LIN {X 0,Y 368.88,Z 241.032,A -85,B 0,C 180,E1 -12741.361,E2 -12741.361} C_VEL
LIN {X 0,Y 368.933,Z 241.028,A -85,B 0,C 180,E1 -12745.14,E2 -12745.14} C_VEL
LIN {X 0,Y 368.915,Z 241.029,A -85,B 0,C 180,E1 -12749.039,E2 -12749.039} C_VEL
LIN {X 0,Y 368.907,Z 241.03,A -85,B 0,C 180,E1 -12751.552,E2 -12751.552} C_VEL
LIN {X 0,Y 368.92,Z 241.03,A -85,B 0,C 180,E1 -12755.216,E2 -12755.216} C_VEL
LIN {X 0,Y 368.917,Z 241.033,A -85,B 0,C 180,E1 -12758.975,E2 -12758.975} C_VEL
LIN {X 0,Y 368.933,Z 241.027,A -85,B 0,C 180,E1 -12762.256,E2 -12762.256} C_VEL
LIN {X 0,Y 369.039,Z 241.014,A -85,B 0,C 180,E1 -12766.216,E2 -12766.216} C_VEL
LIN {X 0,Y 369.049,Z 241.013,A -85,B 0,C 180,E1 -12770.125,E2 -12770.125} C_VEL
LIN {X 0,Y 369.165,Z 240.997,A -85,B 0,C 180,E1 -12773.434,E2 -12773.434} C_VEL
LIN {X 0,Y 369.287,Z 240.984,A -85,B 0,C 180,E1 -12777.812,E2 -12777.812} C_VEL
LIN {X 0,Y 369.437,Z 240.962,A -85,B 0,C 180,E1 -12779.993,E2 -12779.993} C_VEL
LIN {X 0,Y 369.298,Z 240.98,A -85,B 0,C 180,E1 -12782.174,E2 -12782.174} C_VEL
LIN {X 0,Y 369.16,Z 241,A -85,B 0,C 180,E1 -12786.551,E2 -12786.551} C_VEL
LIN {X 0,Y 369.099,Z 241.008,A -85,B 0,C 180,E1 -12788.754,E2 -12788.754} C_VEL
LIN {X 0,Y 368.987,Z 241.022,A -85,B 0,C 180,E1 -12792.086,E2 -12792.086} C_VEL
LIN {X 0,Y 368.969,Z 241.027,A -85,B 0,C 180,E1 -12795.457,E2 -12795.457} C_VEL
LIN {X 0,Y 368.973,Z 241.053,A -85,B 0,C 180,E1 -12799.137,E2 -12799.137} C_VEL
LIN {X 0,Y 369.122,Z 241.853,A -85,B 0,C 180,E1 -12799.454,E2 -12799.454} C_VEL
LIN {X 0,Y 371.497,Z 252.434,A -85,B 0,C 180,E1 -12802.223,E2 -12802.223} C_VEL
LIN {X 0,Y 372.489,Z 258.071,A -85,B 0,C 180,E1 -12803.627,E2 -12803.627} C_VEL
LIN {X 0,Y 372.536,Z 259.043,A -85,B 0,C 180,E1 -12803.809,E2 -12803.809} C_VEL
LIN {X 0,Y 376.937,Z 279.442,A -85,B 0,C 180,E1 -12804.621,E2 -12804.621} C_VEL
LIN {X 0,Y 378.226,Z 287.075,A -85,B 0,C 180,E1 -12804.882,E2 -12804.882} C_VEL
LIN {X 0,Y 376.362,Z 367.62,A -85,B 0,C 180,E1 -12806.593,E2 -12806.593} C_VEL
LIN {X 0,Y 375.694,Z 381.568,A -85,B 0,C 180,E1 -12807.118,E2 -12807.118} C_VEL
LIN {X 0,Y 374.985,Z 393.464,A -85,B 0,C 180,E1 -12807.778,E2 -12807.778} C_VEL
LIN {X 0,Y 374.005,Z 405.344,A -85,B 0,C 180,E1 -12808.66,E2 -12808.66} C_VEL
LIN {X 0,Y 372.898,Z 416.825,A -85,B 0,C 180,E1 -12809.756,E2 -12809.756} C_VEL
LIN {X 0,Y 371.777,Z 427.103,A -85,B 0,C 180,E1 -12810.983,E2 -12810.983} C_VEL
LIN {X 0,Y 370.754,Z 436.401,A -85,B 0,C 180,E1 -12812.367,E2 -12812.367} C_VEL
LIN {X 0,Y 369.821,Z 444.095,A -85,B 0,C 180,E1 -12813.759,E2 -12813.759} C_VEL
LIN {X 0,Y 369.08,Z 450.98,A -85,B 0,C 180,E1 -12815.281,E2 -12815.281} C_VEL
LIN {X 0,Y 368.38,Z 457.744,A -85,B 0,C 180,E1 -12817.156,E2 -12817.156} C_VEL
LIN {X 0,Y 367.823,Z 462.959,A -85,B 0,C 180,E1 -12819.077,E2 -12819.077} C_VEL
LIN {X 0,Y 367.554,Z 465.968,A -85,B 0,C 180,E1 -12820.537,E2 -12820.537} C_VEL
LIN {X 0,Y 367.345,Z 468.186,A -85,B 0,C 180,E1 -12822.024,E2 -12822.024} C_VEL
LIN {X 0,Y 367.242,Z 469.646,A -85,B 0,C 180,E1 -12823.532,E2 -12823.532} C_VEL
LIN {X 0,Y 367.153,Z 470.359,A -85,B 0,C 180,E1 -12825.079,E2 -12825.079} C_VEL
LIN {X 0,Y 367.105,Z 470.265,A -85,B 0,C 180,E1 -12826.661,E2 -12826.661} C_VEL
LIN {X 0,Y 367.181,Z 469.289,A -85,B 0,C 180,E1 -12828.271,E2 -12828.271} C_VEL
LIN {X 0,Y 367.289,Z 467.345,A -85,B 0,C 180,E1 -12829.926,E2 -12829.926} C_VEL
LIN {X 0,Y 367.518,Z 464.352,A -85,B 0,C 180,E1 -12831.615,E2 -12831.615} C_VEL
LIN {X 0,Y 367.894,Z 459.129,A -85,B 0,C 180,E1 -12833.689,E2 -12833.689} C_VEL
LIN {X 0,Y 368.411,Z 453.179,A -85,B 0,C 180,E1 -12835.46,E2 -12835.46} C_VEL
LIN {X 0,Y 368.975,Z 446.012,A -85,B 0,C 180,E1 -12837.149,E2 -12837.149} C_VEL
LIN {X 0,Y 369.786,Z 437.345,A -85,B 0,C 180,E1 -12838.767,E2 -12838.767} C_VEL
LIN {X 0,Y 370.61,Z 428.223,A -85,B 0,C 180,E1 -12840.149,E2 -12840.149} C_VEL
LIN {X 0,Y 371.441,Z 418.859,A -85,B 0,C 180,E1 -12841.309,E2 -12841.309} C_VEL
LIN {X 0,Y 372.382,Z 407.076,A -85,B 0,C 180,E1 -12842.48,E2 -12842.48} C_VEL
LIN {X 0,Y 373.302,Z 394.459,A -85,B 0,C 180,E1 -12843.443,E2 -12843.443} C_VEL
LIN {X 0,Y 373.975,Z 382.071,A -85,B 0,C 180,E1 -12844.149,E2 -12844.149} C_VEL
LIN {X 0,Y 374.556,Z 368.268,A -85,B 0,C 180,E1 -12844.678,E2 -12844.678} C_VEL
LIN {X 0,Y 375.164,Z 336.229,A -85,B 0,C 180,E1 -12845.369,E2 -12845.369} C_VEL
LIN {X 0,Y 376.006,Z 284.873,A -85,B 0,C 180,E1 -12846.423,E2 -12846.423} C_VEL
LIN {X 0,Y 371.483,Z 259.793,A -85,B 0,C 180,E1 -12847.219,E2 -12847.219} C_VEL
LIN {X 0,Y 371.535,Z 258.335,A -85,B 0,C 180,E1 -12847.48,E2 -12847.48} C_VEL
LIN {X 0,Y 371.55,Z 254.8,A -85,B 0,C 180,E1 -12848.409,E2 -12848.409} C_VEL
LIN {X 0,Y 369.334,Z 242.98,A -85,B 0,C 180,E1 -12851.704,E2 -12851.704} C_VEL
LIN {X 0,Y 368.973,Z 241.05,A -85,B 0,C 180,E1 -12852.346,E2 -12852.346} C_VEL
LIN {X 0,Y 368.965,Z 241.024,A -85,B 0,C 180,E1 -12856.227,E2 -12856.227} C_VEL
LIN {X 0,Y 369,Z 241.018,A -85,B 0,C 180,E1 -12860.132,E2 -12860.132} C_VEL
LIN {X 0,Y 369.091,Z 241.008,A -85,B 0,C 180,E1 -12862.342,E2 -12862.342} C_VEL
LIN {X 0,Y 369.078,Z 241.01,A -85,B 0,C 180,E1 -12864.539,E2 -12864.539} C_VEL
LIN {X 0,Y 369.252,Z 240.985,A -85,B 0,C 180,E1 -12867.82,E2 -12867.82} C_VEL
LIN {X 0,Y 369.388,Z 240.968,A -85,B 0,C 180,E1 -12870.002,E2 -12870.002} C_VEL
LIN {X 0,Y 369.088,Z 241.011,A -85,B 0,C 180,E1 -12873.277,E2 -12873.277} C_VEL
LIN {X 0,Y 369.061,Z 241.013,A -85,B 0,C 180,E1 -12873.418,E2 -12873.418} C_VEL
LIN {X 0,Y 368.32,Z 241.102,A -85,B 0,C 180,E1 -12874.329,E2 -12874.329} C_VEL
LIN {X 0,Y 365.557,Z 241.446,A -85,B 0,C 180,E1 -12875.813,E2 -12875.813} C_VEL
LIN {X 0,Y 363.239,Z 241.738,A -85,B 0,C 180,E1 -12877.013,E2 -12877.013} C_VEL
LIN {X 0,Y 362.191,Z 241.866,A -85,B 0,C 180,E1 -12877.939,E2 -12877.939} C_VEL
LIN {X 0,Y 362.073,Z 241.879,A -85,B 0,C 180,E1 -12878.252,E2 -12878.252} C_VEL
LIN {X 0,Y 361.9,Z 241.901,A -85,B 0,C 180,E1 -12882.336,E2 -12882.336} C_VEL
LIN {X 0,Y 361.896,Z 241.901,A -85,B 0,C 180,E1 -12884.625,E2 -12884.625} C_VEL
LIN {X 0,Y 361.892,Z 241.904,A -85,B 0,C 180,E1 -12888.104,E2 -12888.104} C_VEL
LIN {X 0,Y 361.822,Z 241.917,A -85,B 0,C 180,E1 -12891.659,E2 -12891.659} C_VEL
LIN {X 0,Y 361.869,Z 241.906,A -85,B 0,C 180,E1 -12895.296,E2 -12895.296} C_VEL
LIN {X 0,Y 361.866,Z 241.91,A -85,B 0,C 180,E1 -12897.784,E2 -12897.784} C_VEL
LIN {X 0,Y 361.806,Z 241.915,A -85,B 0,C 180,E1 -12901.634,E2 -12901.634} C_VEL
LIN {X 0,Y 361.824,Z 241.91,A -85,B 0,C 180,E1 -12905.352,E2 -12905.352} C_VEL
LIN {X 0,Y 361.827,Z 241.911,A -85,B 0,C 180,E1 -12909.035,E2 -12909.035} C_VEL
LIN {X 0,Y 361.843,Z 241.915,A -85,B 0,C 180,E1 -12912.448,E2 -12912.448} C_VEL
LIN {X 0,Y 361.891,Z 241.903,A -85,B 0,C 180,E1 -12915.937,E2 -12915.937} C_VEL
LIN {X 0,Y 361.87,Z 241.906,A -85,B 0,C 180,E1 -12919.24,E2 -12919.24} C_VEL
LIN {X 0,Y 361.845,Z 241.913,A -85,B 0,C 180,E1 -12922.992,E2 -12922.992} C_VEL
LIN {X 0,Y 361.831,Z 241.913,A -85,B 0,C 180,E1 -12926.64,E2 -12926.64} C_VEL
LIN {X 0,Y 361.849,Z 241.908,A -85,B 0,C 180,E1 -12929.681,E2 -12929.681} C_VEL
LIN {X 0,Y 361.934,Z 241.9,A -85,B 0,C 180,E1 -12933.484,E2 -12933.484} C_VEL
LIN {X 0,Y 361.864,Z 241.911,A -85,B 0,C 180,E1 -12937.153,E2 -12937.153} C_VEL
LIN {X 0,Y 361.872,Z 241.905,A -85,B 0,C 180,E1 -12940.731,E2 -12940.731} C_VEL
LIN {X 0,Y 361.935,Z 241.897,A -85,B 0,C 180,E1 -12944.234,E2 -12944.234} C_VEL
LIN {X 0,Y 361.994,Z 241.889,A -85,B 0,C 180,E1 -12946.536,E2 -12946.536} C_VEL
LIN {X 0,Y 362.026,Z 241.89,A -85,B 0,C 180,E1 -12949.946,E2 -12949.946} C_VEL
LIN {X 0,Y 362.124,Z 241.875,A -85,B 0,C 180,E1 -12953.321,E2 -12953.321} C_VEL
LIN {X 0,Y 362.275,Z 241.859,A -85,B 0,C 180,E1 -12957.784,E2 -12957.784} C_VEL
LIN {X 0,Y 362.271,Z 241.861,A -85,B 0,C 180,E1 -12962.231,E2 -12962.231} C_VEL
LIN {X 0,Y 362.133,Z 241.874,A -85,B 0,C 180,E1 -12966.694,E2 -12966.694} C_VEL
LIN {X 0,Y 362.01,Z 241.89,A -85,B 0,C 180,E1 -12970.069,E2 -12970.069} C_VEL
LIN {X 0,Y 362.015,Z 241.888,A -85,B 0,C 180,E1 -12973.904,E2 -12973.904} C_VEL
LIN {X 0,Y 361.946,Z 241.899,A -85,B 0,C 180,E1 -12976.94,E2 -12976.94} C_VEL
LIN {X 0,Y 361.902,Z 241.904,A -85,B 0,C 180,E1 -12980.466,E2 -12980.466} C_VEL
LIN {X 0,Y 361.915,Z 241.899,A -85,B 0,C 180,E1 -12984.117,E2 -12984.117} C_VEL
LIN {X 0,Y 361.856,Z 241.907,A -85,B 0,C 180,E1 -12987.79,E2 -12987.79} C_VEL
LIN {X 0,Y 361.87,Z 241.91,A -85,B 0,C 180,E1 -12991.289,E2 -12991.289} C_VEL
LIN {X 0,Y 361.876,Z 241.904,A -85,B 0,C 180,E1 -12994.284,E2 -12994.284} C_VEL
LIN {X 0,Y 361.883,Z 241.909,A -85,B 0,C 180,E1 -12997.225,E2 -12997.225} C_VEL
LIN {X 0,Y 361.833,Z 241.91,A -85,B 0,C 180,E1 -13000.753,E2 -13000.753} C_VEL
LIN {X 0,Y 361.81,Z 241.912,A -85,B 0,C 180,E1 -13004.376,E2 -13004.376} C_VEL
LIN {X 0,Y 361.837,Z 241.915,A -85,B 0,C 180,E1 -13007.574,E2 -13007.574} C_VEL
LIN {X 0,Y 361.866,Z 241.909,A -85,B 0,C 180,E1 -13011.573,E2 -13011.573} C_VEL
LIN {X 0,Y 361.894,Z 241.902,A -85,B 0,C 180,E1 -13014.658,E2 -13014.658} C_VEL
LIN {X 0,Y 361.862,Z 241.912,A -85,B 0,C 180,E1 -13018.371,E2 -13018.371} C_VEL
LIN {X 0,Y 361.923,Z 241.987,A -85,B 0,C 180,E1 -13021.432,E2 -13021.432} C_VEL
LIN {X 0,Y 364.248,Z 253.417,A -85,B 0,C 180,E1 -13024.575,E2 -13024.575} C_VEL
LIN {X 0,Y 365.247,Z 259.524,A -85,B 0,C 180,E1 -13026.165,E2 -13026.165} C_VEL
LIN {X 0,Y 364.377,Z 268.912,A -85,B 0,C 180,E1 -13028.396,E2 -13028.396} C_VEL
LIN {X 0,Y 365.363,Z 275.194,A -85,B 0,C 180,E1 -13028.638,E2 -13028.638} C_VEL
LIN {X 0,Y 369.292,Z 299.895,A -85,B 0,C 180,E1 -13029.389,E2 -13029.389} C_VEL
LIN {X 0,Y 367.75,Z 377.611,A -85,B 0,C 180,E1 -13031.04,E2 -13031.04} C_VEL
LIN {X 0,Y 367.12,Z 391.044,A -85,B 0,C 180,E1 -13031.549,E2 -13031.549} C_VEL
LIN {X 0,Y 366.383,Z 403.845,A -85,B 0,C 180,E1 -13032.269,E2 -13032.269} C_VEL
LIN {X 0,Y 365.338,Z 416.379,A -85,B 0,C 180,E1 -13033.227,E2 -13033.227} C_VEL
LIN {X 0,Y 364.389,Z 427.609,A -85,B 0,C 180,E1 -13034.333,E2 -13034.333} C_VEL
LIN {X 0,Y 363.664,Z 436.712,A -85,B 0,C 180,E1 -13035.448,E2 -13035.448} C_VEL
LIN {X 0,Y 362.744,Z 446.03,A -85,B 0,C 180,E1 -13036.839,E2 -13036.839} C_VEL
LIN {X 0,Y 361.838,Z 455.084,A -85,B 0,C 180,E1 -13038.515,E2 -13038.515} C_VEL
LIN {X 0,Y 361.216,Z 462.362,A -85,B 0,C 180,E1 -13040.196,E2 -13040.196} C_VEL
LIN {X 0,Y 360.843,Z 467.262,A -85,B 0,C 180,E1 -13041.599,E2 -13041.599} C_VEL
LIN {X 0,Y 360.529,Z 472.006,A -85,B 0,C 180,E1 -13043.281,E2 -13043.281} C_VEL
LIN {X 0,Y 360.361,Z 475.609,A -85,B 0,C 180,E1 -13044.963,E2 -13044.963} C_VEL
LIN {X 0,Y 360.284,Z 478.174,A -85,B 0,C 180,E1 -13046.643,E2 -13046.643} C_VEL
LIN {X 0,Y 360.234,Z 479.363,A -85,B 0,C 180,E1 -13047.762,E2 -13047.762} C_VEL
LIN {X 0,Y 360.259,Z 480.099,A -85,B 0,C 180,E1 -13048.88,E2 -13048.88} C_VEL
LIN {X 0,Y 360.285,Z 480.438,A -85,B 0,C 180,E1 -13049.998,E2 -13049.998} C_VEL
LIN {X 0,Y 360.257,Z 480.382,A -85,B 0,C 180,E1 -13051.116,E2 -13051.116} C_VEL
LIN {X 0,Y 360.232,Z 479.92,A -85,B 0,C 180,E1 -13052.234,E2 -13052.234} C_VEL
LIN {X 0,Y 360.284,Z 479.017,A -85,B 0,C 180,E1 -13053.353,E2 -13053.353} C_VEL
LIN {X 0,Y 360.37,Z 477.711,A -85,B 0,C 180,E1 -13054.472,E2 -13054.472} C_VEL
LIN {X 0,Y 360.474,Z 475.098,A -85,B 0,C 180,E1 -13056.076,E2 -13056.076} C_VEL
LIN {X 0,Y 360.771,Z 471.152,A -85,B 0,C 180,E1 -13057.835,E2 -13057.835} C_VEL
LIN {X 0,Y 361.265,Z 466.224,A -85,B 0,C 180,E1 -13059.516,E2 -13059.516} C_VEL
LIN {X 0,Y 361.94,Z 460.024,A -85,B 0,C 180,E1 -13061.194,E2 -13061.194} C_VEL
LIN {X 0,Y 362.832,Z 452.335,A -85,B 0,C 180,E1 -13062.869,E2 -13062.869} C_VEL
LIN {X 0,Y 364.083,Z 442.682,A -85,B 0,C 180,E1 -13064.531,E2 -13064.531} C_VEL
LIN {X 0,Y 365.093,Z 432.754,A -85,B 0,C 180,E1 -13065.919,E2 -13065.919} C_VEL
LIN {X 0,Y 366.141,Z 423.009,A -85,B 0,C 180,E1 -13067.019,E2 -13067.019} C_VEL
LIN {X 0,Y 367.4,Z 410.731,A -85,B 0,C 180,E1 -13068.108,E2 -13068.108} C_VEL
LIN {X 0,Y 368.393,Z 399.904,A -85,B 0,C 180,E1 -13068.85,E2 -13068.85} C_VEL
LIN {X 0,Y 369.213,Z 386.728,A -85,B 0,C 180,E1 -13069.528,E2 -13069.528} C_VEL
LIN {X 0,Y 369.858,Z 373.38,A -85,B 0,C 180,E1 -13069.962,E2 -13069.962} C_VEL
LIN {X 0,Y 371.447,Z 299.693,A -85,B 0,C 180,E1 -13071.55,E2 -13071.55} C_VEL
LIN {X 0,Y 367.766,Z 278.61,A -85,B 0,C 180,E1 -13072.318,E2 -13072.318} C_VEL
LIN {X 0,Y 365.474,Z 268.168,A -85,B 0,C 180,E1 -13072.764,E2 -13072.764} C_VEL
LIN {X 0,Y 365.983,Z 262.373,A -85,B 0,C 180,E1 -13074.081,E2 -13074.081} C_VEL
LIN {X 0,Y 364.601,Z 253.875,A -85,B 0,C 180,E1 -13076.315,E2 -13076.315} C_VEL
LIN {X 0,Y 362.372,Z 244.187,A -85,B 0,C 180,E1 -13079.001,E2 -13079.001} C_VEL
LIN {X 0,Y 361.899,Z 241.952,A -85,B 0,C 180,E1 -13079.72,E2 -13079.72} C_VEL
LIN {X 0,Y 361.87,Z 241.91,A -85,B 0,C 180,E1 -13083.365,E2 -13083.365} C_VEL
LIN {X 0,Y 361.873,Z 241.909,A -85,B 0,C 180,E1 -13087.014,E2 -13087.014} C_VEL
LIN {X 0,Y 361.819,Z 241.913,A -85,B 0,C 180,E1 -13090.746,E2 -13090.746} C_VEL
LIN {X 0,Y 361.818,Z 241.917,A -85,B 0,C 180,E1 -13094.365,E2 -13094.365} C_VEL
LIN {X 0,Y 361.828,Z 241.913,A -85,B 0,C 180,E1 -13097.566,E2 -13097.566} C_VEL
LIN {X 0,Y 361.846,Z 241.909,A -85,B 0,C 180,E1 -13101.566,E2 -13101.566} C_VEL
LIN {X 0,Y 361.873,Z 241.909,A -85,B 0,C 180,E1 -13104.651,E2 -13104.651} C_VEL
LIN {X 0,Y 361.84,Z 241.914,A -85,B 0,C 180,E1 -13108.365,E2 -13108.365} C_VEL
LIN {X 0,Y 361.85,Z 241.91,A -85,B 0,C 180,E1 -13110.945,E2 -13110.945} C_VEL
LIN {X 0,Y 361.878,Z 241.906,A -85,B 0,C 180,E1 -13114.7,E2 -13114.7} C_VEL
LIN {X 0,Y 361.85,Z 241.908,A -85,B 0,C 180,E1 -13118.338,E2 -13118.338} C_VEL
LIN {X 0,Y 361.89,Z 241.903,A -85,B 0,C 180,E1 -13122.091,E2 -13122.091} C_VEL
LIN {X 0,Y 361.98,Z 241.894,A -85,B 0,C 180,E1 -13126.102,E2 -13126.102} C_VEL
LIN {X 0,Y 361.986,Z 241.893,A -85,B 0,C 180,E1 -13129.93,E2 -13129.93} C_VEL
LIN {X 0,Y 362.127,Z 241.875,A -85,B 0,C 180,E1 -13133.306,E2 -13133.306} C_VEL
LIN {X 0,Y 362.25,Z 241.86,A -85,B 0,C 180,E1 -13137.769,E2 -13137.769} C_VEL
LIN {X 0,Y 362.386,Z 241.84,A -85,B 0,C 180,E1 -13139.993,E2 -13139.993} C_VEL
LIN {X 0,Y 362.261,Z 241.856,A -85,B 0,C 180,E1 -13142.216,E2 -13142.216} C_VEL
LIN {X 0,Y 362.124,Z 241.877,A -85,B 0,C 180,E1 -13146.679,E2 -13146.679} C_VEL
LIN {X 0,Y 362.011,Z 241.891,A -85,B 0,C 180,E1 -13150.054,E2 -13150.054} C_VEL
LIN {X 0,Y 361.97,Z 241.898,A -85,B 0,C 180,E1 -13153.892,E2 -13153.892} C_VEL
LIN {X 0,Y 361.938,Z 241.899,A -85,B 0,C 180,E1 -13157.933,E2 -13157.933} C_VEL
LIN {X 0,Y 361.962,Z 242.037,A -85,B 0,C 180,E1 -13158.75,E2 -13158.75} C_VEL
LIN {X 0,Y 364.246,Z 252.021,A -85,B 0,C 180,E1 -13161.497,E2 -13161.497} C_VEL
LIN {X 0,Y 365.659,Z 258.999,A -85,B 0,C 180,E1 -13163.27,E2 -13163.27} C_VEL
LIN {X 0,Y 367.677,Z 267.137,A -85,B 0,C 180,E1 -13163.657,E2 -13163.657} C_VEL
LIN {X 0,Y 371.681,Z 286.962,A -85,B 0,C 180,E1 -13164.423,E2 -13164.423} C_VEL
LIN {X 0,Y 369.795,Z 367.824,A -85,B 0,C 180,E1 -13166.183,E2 -13166.183} C_VEL
LIN {X 0,Y 369.116,Z 381.433,A -85,B 0,C 180,E1 -13166.703,E2 -13166.703} C_VEL
LIN {X 0,Y 368.336,Z 393.75,A -85,B 0,C 180,E1 -13167.397,E2 -13167.397} C_VEL
LIN {X 0,Y 367.268,Z 406.035,A -85,B 0,C 180,E1 -13168.333,E2 -13168.333} C_VEL
LIN {X 0,Y 366.128,Z 417.468,A -85,B 0,C 180,E1 -13169.454,E2 -13169.454} C_VEL
LIN {X 0,Y 364.962,Z 427.464,A -85,B 0,C 180,E1 -13170.68,E2 -13170.68} C_VEL
LIN {X 0,Y 363.751,Z 437.747,A -85,B 0,C 180,E1 -13172.265,E2 -13172.265} C_VEL
LIN {X 0,Y 362.704,Z 446.064,A -85,B 0,C 180,E1 -13173.857,E2 -13173.857} C_VEL
LIN {X 0,Y 361.852,Z 453.395,A -85,B 0,C 180,E1 -13175.627,E2 -13175.627} C_VEL
LIN {X 0,Y 361.303,Z 458.357,A -85,B 0,C 180,E1 -13177.11,E2 -13177.11} C_VEL
LIN {X 0,Y 360.789,Z 462.891,A -85,B 0,C 180,E1 -13178.818,E2 -13178.818} C_VEL
LIN {X 0,Y 360.463,Z 466.266,A -85,B 0,C 180,E1 -13180.505,E2 -13180.505} C_VEL
LIN {X 0,Y 360.25,Z 468.601,A -85,B 0,C 180,E1 -13182.159,E2 -13182.159} C_VEL
LIN {X 0,Y 360.121,Z 469.991,A -85,B 0,C 180,E1 -13183.777,E2 -13183.777} C_VEL
LIN {X 0,Y 360.043,Z 470.506,A -85,B 0,C 180,E1 -13185.358,E2 -13185.358} C_VEL
LIN {X 0,Y 360.018,Z 470.24,A -85,B 0,C 180,E1 -13186.906,E2 -13186.906} C_VEL
LIN {X 0,Y 360.083,Z 469.235,A -85,B 0,C 180,E1 -13188.428,E2 -13188.428} C_VEL
LIN {X 0,Y 360.295,Z 466.376,A -85,B 0,C 180,E1 -13190.629,E2 -13190.629} C_VEL
LIN {X 0,Y 360.625,Z 461.794,A -85,B 0,C 180,E1 -13192.836,E2 -13192.836} C_VEL
LIN {X 0,Y 361.112,Z 456.042,A -85,B 0,C 180,E1 -13194.808,E2 -13194.808} C_VEL
LIN {X 0,Y 361.719,Z 449.081,A -85,B 0,C 180,E1 -13196.645,E2 -13196.645} C_VEL
LIN {X 0,Y 362.308,Z 442.248,A -85,B 0,C 180,E1 -13198.092,E2 -13198.092} C_VEL
LIN {X 0,Y 363.179,Z 433.295,A -85,B 0,C 180,E1 -13199.635,E2 -13199.635} C_VEL
LIN {X 0,Y 364.096,Z 423.384,A -85,B 0,C 180,E1 -13201.02,E2 -13201.02} C_VEL
LIN {X 0,Y 365.122,Z 412.051,A -85,B 0,C 180,E1 -13202.28,E2 -13202.28} C_VEL
LIN {X 0,Y 366.059,Z 399.91,A -85,B 0,C 180,E1 -13203.337,E2 -13203.337} C_VEL
LIN {X 0,Y 366.872,Z 387.097,A -85,B 0,C 180,E1 -13204.18,E2 -13204.18} C_VEL
LIN {X 0,Y 367.518,Z 373.473,A -85,B 0,C 180,E1 -13204.808,E2 -13204.808} C_VEL
LIN {X 0,Y 367.969,Z 359.673,A -85,B 0,C 180,E1 -13205.197,E2 -13205.197} C_VEL
LIN {X 0,Y 369.272,Z 285.9,A -85,B 0,C 180,E1 -13206.742,E2 -13206.742} C_VEL
LIN {X 0,Y 364.621,Z 260.016,A -85,B 0,C 180,E1 -13207.573,E2 -13207.573} C_VEL
LIN {X 0,Y 364.641,Z 258.567,A -85,B 0,C 180,E1 -13207.82,E2 -13207.82} C_VEL
LIN {X 0,Y 364.184,Z 253.951,A -85,B 0,C 180,E1 -13209.086,E2 -13209.086} C_VEL
LIN {X 0,Y 361.936,Z 242.118,A -85,B 0,C 180,E1 -13212.486,E2 -13212.486} C_VEL
LIN {X 0,Y 361.926,Z 241.9,A -85,B 0,C 180,E1 -13216.101,E2 -13216.101} C_VEL
LIN {X 0,Y 361.964,Z 241.893,A -85,B 0,C 180,E1 -13219.938,E2 -13219.938} C_VEL
LIN {X 0,Y 362.095,Z 241.878,A -85,B 0,C 180,E1 -13223.314,E2 -13223.314} C_VEL
LIN {X 0,Y 362.218,Z 241.861,A -85,B 0,C 180,E1 -13227.778,E2 -13227.778} C_VEL
LIN {X 0,Y 362.358,Z 241.844,A -85,B 0,C 180,E1 -13230.002,E2 -13230.002} C_VEL
LIN {X 0,Y 362.218,Z 241.861,A -85,B 0,C 180,E1 -13232.226,E2 -13232.226} C_VEL
LIN {X 0,Y 362.098,Z 241.878,A -85,B 0,C 180,E1 -13236.689,E2 -13236.689} C_VEL
LIN {X 0,Y 362.073,Z 241.879,A -85,B 0,C 180,E1 -13238.252,E2 -13238.252} C_VEL
LIN {X 0,Y 361.302,Z 241.981,A -85,B 0,C 180,E1 -13239.18,E2 -13239.18} C_VEL
LIN {X 0,Y 358.365,Z 242.342,A -85,B 0,C 180,E1 -13240.688,E2 -13240.688} C_VEL
LIN {X 0,Y 355.945,Z 242.645,A -85,B 0,C 180,E1 -13241.908,E2 -13241.908} C_VEL
LIN {X 0,Y 354.928,Z 242.771,A -85,B 0,C 180,E1 -13242.853,E2 -13242.853} C_VEL
LIN {X 0,Y 354.854,Z 242.778,A -85,B 0,C 180,E1 -13243.173,E2 -13243.173} C_VEL
LIN {X 0,Y 354.824,Z 242.784,A -85,B 0,C 180,E1 -13246.101,E2 -13246.101} C_VEL
LIN {X 0,Y 354.837,Z 242.781,A -85,B 0,C 180,E1 -13248.477,E2 -13248.477} C_VEL
LIN {X 0,Y 354.769,Z 242.792,A -85,B 0,C 180,E1 -13252.112,E2 -13252.112} C_VEL
LIN {X 0,Y 354.841,Z 242.787,A -85,B 0,C 180,E1 -13255.834,E2 -13255.834} C_VEL
LIN {X 0,Y 354.8,Z 242.789,A -85,B 0,C 180,E1 -13259.685,E2 -13259.685} C_VEL
LIN {X 0,Y 354.78,Z 242.79,A -85,B 0,C 180,E1 -13263.689,E2 -13263.689} C_VEL
LIN {X 0,Y 354.75,Z 242.796,A -85,B 0,C 180,E1 -13266.467,E2 -13266.467} C_VEL
LIN {X 0,Y 354.779,Z 242.788,A -85,B 0,C 180,E1 -13269.431,E2 -13269.431} C_VEL
LIN {X 0,Y 354.799,Z 242.788,A -85,B 0,C 180,E1 -13272.884,E2 -13272.884} C_VEL
LIN {X 0,Y 354.829,Z 242.784,A -85,B 0,C 180,E1 -13276.127,E2 -13276.127} C_VEL
LIN {X 0,Y 354.821,Z 242.784,A -85,B 0,C 180,E1 -13279.197,E2 -13279.197} C_VEL
LIN {X 0,Y 354.784,Z 242.79,A -85,B 0,C 180,E1 -13282.41,E2 -13282.41} C_VEL
LIN {X 0,Y 354.784,Z 242.794,A -85,B 0,C 180,E1 -13284.95,E2 -13284.95} C_VEL
LIN {X 0,Y 354.768,Z 242.791,A -85,B 0,C 180,E1 -13288.414,E2 -13288.414} C_VEL
LIN {X 0,Y 354.825,Z 242.784,A -85,B 0,C 180,E1 -13291.627,E2 -13291.627} C_VEL
LIN {X 0,Y 354.88,Z 242.775,A -85,B 0,C 180,E1 -13294.181,E2 -13294.181} C_VEL
LIN {X 0,Y 354.801,Z 242.786,A -85,B 0,C 180,E1 -13297.901,E2 -13297.901} C_VEL
LIN {X 0,Y 354.88,Z 242.777,A -85,B 0,C 180,E1 -13301.917,E2 -13301.917} C_VEL
LIN {X 0,Y 354.937,Z 242.771,A -85,B 0,C 180,E1 -13305.99,E2 -13305.99} C_VEL
LIN {X 0,Y 354.973,Z 242.771,A -85,B 0,C 180,E1 -13309.744,E2 -13309.744} C_VEL
LIN {X 0,Y 355.09,Z 242.75,A -85,B 0,C 180,E1 -13313.188,E2 -13313.188} C_VEL
LIN {X 0,Y 355.238,Z 242.735,A -85,B 0,C 180,E1 -13317.74,E2 -13317.74} C_VEL
LIN {X 0,Y 355.176,Z 242.739,A -85,B 0,C 180,E1 -13321.141,E2 -13321.141} C_VEL
LIN {X 0,Y 355.234,Z 242.737,A -85,B 0,C 180,E1 -13322.275,E2 -13322.275} C_VEL
LIN {X 0,Y 355.099,Z 242.75,A -85,B 0,C 180,E1 -13326.827,E2 -13326.827} C_VEL
LIN {X 0,Y 354.967,Z 242.77,A -85,B 0,C 180,E1 -13330.271,E2 -13330.271} C_VEL
LIN {X 0,Y 354.959,Z 242.767,A -85,B 0,C 180,E1 -13334.024,E2 -13334.024} C_VEL
LIN {X 0,Y 354.909,Z 242.773,A -85,B 0,C 180,E1 -13338.098,E2 -13338.098} C_VEL
LIN {X 0,Y 354.833,Z 242.782,A -85,B 0,C 180,E1 -13342.113,E2 -13342.113} C_VEL
LIN {X 0,Y 354.869,Z 242.78,A -85,B 0,C 180,E1 -13344.582,E2 -13344.582} C_VEL
LIN {X 0,Y 354.819,Z 242.784,A -85,B 0,C 180,E1 -13348.39,E2 -13348.39} C_VEL
LIN {X 0,Y 354.809,Z 242.784,A -85,B 0,C 180,E1 -13352.337,E2 -13352.337} C_VEL
LIN {X 0,Y 354.844,Z 242.782,A -85,B 0,C 180,E1 -13355.702,E2 -13355.702} C_VEL
LIN {X 0,Y 354.793,Z 242.793,A -85,B 0,C 180,E1 -13359.415,E2 -13359.415} C_VEL
LIN {X 0,Y 354.785,Z 242.788,A -85,B 0,C 180,E1 -13362.865,E2 -13362.865} C_VEL
LIN {X 0,Y 354.768,Z 242.791,A -85,B 0,C 180,E1 -13366.102,E2 -13366.102} C_VEL
LIN {X 0,Y 354.785,Z 242.789,A -85,B 0,C 180,E1 -13369.177,E2 -13369.177} C_VEL
LIN {X 0,Y 354.823,Z 242.784,A -85,B 0,C 180,E1 -13372.406,E2 -13372.406} C_VEL
LIN {X 0,Y 354.832,Z 242.781,A -85,B 0,C 180,E1 -13374.941,E2 -13374.941} C_VEL
LIN {X 0,Y 354.818,Z 242.79,A -85,B 0,C 180,E1 -13378.406,E2 -13378.406} C_VEL
LIN {X 0,Y 354.884,Z 242.917,A -85,B 0,C 180,E1 -13381.167,E2 -13381.167} C_VEL
LIN {X 0,Y 357.197,Z 254.28,A -85,B 0,C 180,E1 -13384.349,E2 -13384.349} C_VEL
LIN {X 0,Y 358.252,Z 260.391,A -85,B 0,C 180,E1 -13385.978,E2 -13385.978} C_VEL
LIN {X 0,Y 357.499,Z 268.825,A -85,B 0,C 180,E1 -13388.023,E2 -13388.023} C_VEL
LIN {X 0,Y 359.02,Z 278.379,A -85,B 0,C 180,E1 -13388.369,E2 -13388.369} C_VEL
LIN {X 0,Y 362.548,Z 300.61,A -85,B 0,C 180,E1 -13389.062,E2 -13389.062} C_VEL
LIN {X 0,Y 360.955,Z 376.817,A -85,B 0,C 180,E1 -13390.706,E2 -13390.706} C_VEL
LIN {X 0,Y 360.321,Z 390.465,A -85,B 0,C 180,E1 -13391.225,E2 -13391.225} C_VEL
LIN {X 0,Y 359.564,Z 402.895,A -85,B 0,C 180,E1 -13391.922,E2 -13391.922} C_VEL
LIN {X 0,Y 358.665,Z 414.041,A -85,B 0,C 180,E1 -13392.758,E2 -13392.758} C_VEL
LIN {X 0,Y 357.651,Z 425.676,A -85,B 0,C 180,E1 -13393.883,E2 -13393.883} C_VEL
LIN {X 0,Y 356.761,Z 436.177,A -85,B 0,C 180,E1 -13395.16,E2 -13395.16} C_VEL
LIN {X 0,Y 355.787,Z 445.597,A -85,B 0,C 180,E1 -13396.577,E2 -13396.577} C_VEL
LIN {X 0,Y 354.846,Z 454.711,A -85,B 0,C 180,E1 -13398.285,E2 -13398.285} C_VEL
LIN {X 0,Y 354.193,Z 462.046,A -85,B 0,C 180,E1 -13400,E2 -13400} C_VEL
LIN {X 0,Y 353.802,Z 466.985,A -85,B 0,C 180,E1 -13401.43,E2 -13401.43} C_VEL
LIN {X 0,Y 353.446,Z 471.769,A -85,B 0,C 180,E1 -13403.146,E2 -13403.146} C_VEL
LIN {X 0,Y 353.268,Z 475.408,A -85,B 0,C 180,E1 -13404.862,E2 -13404.862} C_VEL
LIN {X 0,Y 353.208,Z 478.007,A -85,B 0,C 180,E1 -13406.576,E2 -13406.576} C_VEL
LIN {X 0,Y 353.145,Z 479.22,A -85,B 0,C 180,E1 -13407.717,E2 -13407.717} C_VEL
LIN {X 0,Y 353.158,Z 479.978,A -85,B 0,C 180,E1 -13408.858,E2 -13408.858} C_VEL
LIN {X 0,Y 353.186,Z 480.331,A -85,B 0,C 180,E1 -13409.998,E2 -13409.998} C_VEL
LIN {X 0,Y 353.157,Z 480.289,A -85,B 0,C 180,E1 -13411.138,E2 -13411.138} C_VEL
LIN {X 0,Y 353.143,Z 479.849,A -85,B 0,C 180,E1 -13412.279,E2 -13412.279} C_VEL
LIN {X 0,Y 353.209,Z 478.964,A -85,B 0,C 180,E1 -13413.42,E2 -13413.42} C_VEL
LIN {X 0,Y 353.287,Z 477.671,A -85,B 0,C 180,E1 -13414.562,E2 -13414.562} C_VEL
LIN {X 0,Y 353.389,Z 475.372,A -85,B 0,C 180,E1 -13416.048,E2 -13416.048} C_VEL
LIN {X 0,Y 353.726,Z 471.178,A -85,B 0,C 180,E1 -13417.992,E2 -13417.992} C_VEL
LIN {X 0,Y 354.231,Z 466.293,A -85,B 0,C 180,E1 -13419.707,E2 -13419.707} C_VEL
LIN {X 0,Y 354.938,Z 460.14,A -85,B 0,C 180,E1 -13421.418,E2 -13421.418} C_VEL
LIN {X 0,Y 355.919,Z 452.498,A -85,B 0,C 180,E1 -13423.123,E2 -13423.123} C_VEL
LIN {X 0,Y 357.004,Z 444.693,A -85,B 0,C 180,E1 -13424.534,E2 -13424.534} C_VEL
LIN {X 0,Y 358.035,Z 435.188,A -85,B 0,C 180,E1 -13425.949,E2 -13425.949} C_VEL
LIN {X 0,Y 359.253,Z 424.67,A -85,B 0,C 180,E1 -13427.209,E2 -13427.209} C_VEL
LIN {X 0,Y 360.569,Z 412.998,A -85,B 0,C 180,E1 -13428.316,E2 -13428.316} C_VEL
LIN {X 0,Y 361.574,Z 401.726,A -85,B 0,C 180,E1 -13429.145,E2 -13429.145} C_VEL
LIN {X 0,Y 362.572,Z 387.774,A -85,B 0,C 180,E1 -13429.901,E2 -13429.901} C_VEL
LIN {X 0,Y 363.237,Z 375.474,A -85,B 0,C 180,E1 -13430.342,E2 -13430.342} C_VEL
LIN {X 0,Y 365.02,Z 300.893,A -85,B 0,C 180,E1 -13431.992,E2 -13431.992} C_VEL
LIN {X 0,Y 361.842,Z 282.186,A -85,B 0,C 180,E1 -13432.685,E2 -13432.685} C_VEL
LIN {X 0,Y 358.768,Z 267.831,A -85,B 0,C 180,E1 -13433.327,E2 -13433.327} C_VEL
LIN {X 0,Y 359.017,Z 262.654,A -85,B 0,C 180,E1 -13434.579,E2 -13434.579} C_VEL
LIN {X 0,Y 357.117,Z 252.395,A -85,B 0,C 180,E1 -13437.371,E2 -13437.371} C_VEL
LIN {X 0,Y 354.842,Z 242.847,A -85,B 0,C 180,E1 -13440.209,E2 -13440.209} C_VEL
LIN {X 0,Y 354.819,Z 242.789,A -85,B 0,C 180,E1 -13443.698,E2 -13443.698} C_VEL
LIN {X 0,Y 354.806,Z 242.791,A -85,B 0,C 180,E1 -13446.456,E2 -13446.456} C_VEL
LIN {X 0,Y 354.779,Z 242.791,A -85,B 0,C 180,E1 -13449.408,E2 -13449.408} C_VEL
LIN {X 0,Y 354.789,Z 242.788,A -85,B 0,C 180,E1 -13452.861,E2 -13452.861} C_VEL
LIN {X 0,Y 354.768,Z 242.792,A -85,B 0,C 180,E1 -13456.097,E2 -13456.097} C_VEL
LIN {X 0,Y 354.768,Z 242.793,A -85,B 0,C 180,E1 -13459.17,E2 -13459.17} C_VEL
LIN {X 0,Y 354.803,Z 242.791,A -85,B 0,C 180,E1 -13462.399,E2 -13462.399} C_VEL
LIN {X 0,Y 354.811,Z 242.789,A -85,B 0,C 180,E1 -13464.934,E2 -13464.934} C_VEL
LIN {X 0,Y 354.796,Z 242.792,A -85,B 0,C 180,E1 -13468.399,E2 -13468.399} C_VEL
LIN {X 0,Y 354.789,Z 242.789,A -85,B 0,C 180,E1 -13471.607,E2 -13471.607} C_VEL
LIN {X 0,Y 354.841,Z 242.783,A -85,B 0,C 180,E1 -13475.416,E2 -13475.416} C_VEL
LIN {X 0,Y 354.815,Z 242.788,A -85,B 0,C 180,E1 -13479.106,E2 -13479.106} C_VEL
LIN {X 0,Y 354.833,Z 242.787,A -85,B 0,C 180,E1 -13482.71,E2 -13482.71} C_VEL
LIN {X 0,Y 354.939,Z 242.771,A -85,B 0,C 180,E1 -13486.248,E2 -13486.248} C_VEL
LIN {X 0,Y 354.943,Z 242.771,A -85,B 0,C 180,E1 -13489.728,E2 -13489.728} C_VEL
LIN {X 0,Y 355.091,Z 242.753,A -85,B 0,C 180,E1 -13493.173,E2 -13493.173} C_VEL
LIN {X 0,Y 355.213,Z 242.736,A -85,B 0,C 180,E1 -13497.725,E2 -13497.725} C_VEL
LIN {X 0,Y 355.336,Z 242.718,A -85,B 0,C 180,E1 -13499.993,E2 -13499.993} C_VEL
LIN {X 0,Y 355.224,Z 242.733,A -85,B 0,C 180,E1 -13502.26,E2 -13502.26} C_VEL
LIN {X 0,Y 355.09,Z 242.753,A -85,B 0,C 180,E1 -13506.812,E2 -13506.812} C_VEL
LIN {X 0,Y 354.958,Z 242.769,A -85,B 0,C 180,E1 -13510.256,E2 -13510.256} C_VEL
LIN {X 0,Y 354.915,Z 242.777,A -85,B 0,C 180,E1 -13514.012,E2 -13514.012} C_VEL
LIN {X 0,Y 354.914,Z 242.876,A -85,B 0,C 180,E1 -13518.214,E2 -13518.214} C_VEL
LIN {X 0,Y 357.207,Z 252.764,A -85,B 0,C 180,E1 -13521.033,E2 -13521.033} C_VEL
LIN {X 0,Y 358.569,Z 259.336,A -85,B 0,C 180,E1 -13522.723,E2 -13522.723} C_VEL
LIN {X 0,Y 360.426,Z 264.571,A -85,B 0,C 180,E1 -13523.02,E2 -13523.02} C_VEL
LIN {X 0,Y 364.798,Z 285.505,A -85,B 0,C 180,E1 -13523.876,E2 -13523.876} C_VEL
LIN {X 0,Y 365.282,Z 289.608,A -85,B 0,C 180,E1 -13524.011,E2 -13524.011} C_VEL
LIN {X 0,Y 363.266,Z 368.071,A -85,B 0,C 180,E1 -13525.756,E2 -13525.756} C_VEL
LIN {X 0,Y 362.524,Z 381.844,A -85,B 0,C 180,E1 -13526.295,E2 -13526.295} C_VEL
LIN {X 0,Y 361.695,Z 394.113,A -85,B 0,C 180,E1 -13527.007,E2 -13527.007} C_VEL
LIN {X 0,Y 360.715,Z 405.301,A -85,B 0,C 180,E1 -13527.868,E2 -13527.868} C_VEL
LIN {X 0,Y 359.629,Z 415.405,A -85,B 0,C 180,E1 -13528.844,E2 -13528.844} C_VEL
LIN {X 0,Y 358.275,Z 426.752,A -85,B 0,C 180,E1 -13530.215,E2 -13530.215} C_VEL
LIN {X 0,Y 357.2,Z 435.764,A -85,B 0,C 180,E1 -13531.58,E2 -13531.58} C_VEL
LIN {X 0,Y 356.011,Z 444.468,A -85,B 0,C 180,E1 -13533.205,E2 -13533.205} C_VEL
LIN {X 0,Y 355.044,Z 452.243,A -85,B 0,C 180,E1 -13535.021,E2 -13535.021} C_VEL
LIN {X 0,Y 354.278,Z 458.724,A -85,B 0,C 180,E1 -13536.97,E2 -13536.97} C_VEL
LIN {X 0,Y 353.781,Z 462.91,A -85,B 0,C 180,E1 -13538.584,E2 -13538.584} C_VEL
LIN {X 0,Y 353.439,Z 466.117,A -85,B 0,C 180,E1 -13540.187,E2 -13540.187} C_VEL
LIN {X 0,Y 353.27,Z 467.427,A -85,B 0,C 180,E1 -13541.02,E2 -13541.02} C_VEL
LIN {X 0,Y 353.125,Z 469.241,A -85,B 0,C 180,E1 -13542.579,E2 -13542.579} C_VEL
LIN {X 0,Y 352.996,Z 470.336,A -85,B 0,C 180,E1 -13544.217,E2 -13544.217} C_VEL
LIN {X 0,Y 352.943,Z 470.608,A -85,B 0,C 180,E1 -13545.822,E2 -13545.822} C_VEL
LIN {X 0,Y 352.945,Z 470.077,A -85,B 0,C 180,E1 -13547.441,E2 -13547.441} C_VEL
LIN {X 0,Y 353.027,Z 468.61,A -85,B 0,C 180,E1 -13549.14,E2 -13549.14} C_VEL
LIN {X 0,Y 353.244,Z 466.147,A -85,B 0,C 180,E1 -13550.872,E2 -13550.872} C_VEL
LIN {X 0,Y 353.496,Z 462.524,A -85,B 0,C 180,E1 -13552.662,E2 -13552.662} C_VEL
LIN {X 0,Y 353.915,Z 457.559,A -85,B 0,C 180,E1 -13554.487,E2 -13554.487} C_VEL
LIN {X 0,Y 354.513,Z 450.992,A -85,B 0,C 180,E1 -13556.35,E2 -13556.35} C_VEL
LIN {X 0,Y 355.16,Z 443.633,A -85,B 0,C 180,E1 -13558.015,E2 -13558.015} C_VEL
LIN {X 0,Y 355.915,Z 436.227,A -85,B 0,C 180,E1 -13559.385,E2 -13559.385} C_VEL
LIN {X 0,Y 356.86,Z 426.731,A -85,B 0,C 180,E1 -13560.831,E2 -13560.831} C_VEL
LIN {X 0,Y 357.939,Z 415.354,A -85,B 0,C 180,E1 -13562.207,E2 -13562.207} C_VEL
LIN {X 0,Y 358.92,Z 403.548,A -85,B 0,C 180,E1 -13563.336,E2 -13563.336} C_VEL
LIN {X 0,Y 359.819,Z 391.026,A -85,B 0,C 180,E1 -13564.244,E2 -13564.244} C_VEL
LIN {X 0,Y 360.536,Z 378.028,A -85,B 0,C 180,E1 -13564.936,E2 -13564.936} C_VEL
LIN {X 0,Y 361.035,Z 365.517,A -85,B 0,C 180,E1 -13565.376,E2 -13565.376} C_VEL
LIN {X 0,Y 362.471,Z 286.44,A -85,B 0,C 180,E1 -13567.083,E2 -13567.083} C_VEL
LIN {X 0,Y 357.73,Z 259.745,A -85,B 0,C 180,E1 -13567.977,E2 -13567.977} C_VEL
LIN {X 0,Y 357.347,Z 255.963,A -85,B 0,C 180,E1 -13568.968,E2 -13568.968} C_VEL
LIN {X 0,Y 355.191,Z 244.507,A -85,B 0,C 180,E1 -13572.291,E2 -13572.291} C_VEL
LIN {X 0,Y 354.851,Z 242.812,A -85,B 0,C 180,E1 -13572.868,E2 -13572.868} C_VEL
LIN {X 0,Y 354.88,Z 242.779,A -85,B 0,C 180,E1 -13576.255,E2 -13576.255} C_VEL
LIN {X 0,Y 354.911,Z 242.772,A -85,B 0,C 180,E1 -13579.736,E2 -13579.736} C_VEL
LIN {X 0,Y 355.059,Z 242.756,A -85,B 0,C 180,E1 -13583.181,E2 -13583.181} C_VEL
LIN {X 0,Y 355.182,Z 242.738,A -85,B 0,C 180,E1 -13587.734,E2 -13587.734} C_VEL
LIN {X 0,Y 355.328,Z 242.72,A -85,B 0,C 180,E1 -13590.002,E2 -13590.002} C_VEL
LIN {X 0,Y 355.183,Z 242.738,A -85,B 0,C 180,E1 -13592.27,E2 -13592.27} C_VEL
LIN {X 0,Y 355.061,Z 242.755,A -85,B 0,C 180,E1 -13596.823,E2 -13596.823} C_VEL
LIN {X 0,Y 354.915,Z 242.771,A -85,B 0,C 180,E1 -13600.268,E2 -13600.268} C_VEL
LIN {X 0,Y 354.854,Z 242.778,A -85,B 0,C 180,E1 -13603.173,E2 -13603.173} C_VEL
LIN {X 0,Y 354.199,Z 242.864,A -85,B 0,C 180,E1 -13604.121,E2 -13604.121} C_VEL
LIN {X 0,Y 351.32,Z 243.226,A -85,B 0,C 180,E1 -13605.661,E2 -13605.661} C_VEL
LIN {X 0,Y 348.893,Z 243.528,A -85,B 0,C 180,E1 -13606.908,E2 -13606.908} C_VEL
LIN {X 0,Y 347.885,Z 243.651,A -85,B 0,C 180,E1 -13607.874,E2 -13607.874} C_VEL
LIN {X 0,Y 347.821,Z 243.656,A -85,B 0,C 180,E1 -13608.201,E2 -13608.201} C_VEL
LIN {X 0,Y 347.716,Z 243.673,A -85,B 0,C 180,E1 -13611.636,E2 -13611.636} C_VEL
LIN {X 0,Y 347.753,Z 243.664,A -85,B 0,C 180,E1 -13615.115,E2 -13615.115} C_VEL
LIN {X 0,Y 347.756,Z 243.667,A -85,B 0,C 180,E1 -13617.7,E2 -13617.7} C_VEL
LIN {X 0,Y 347.716,Z 243.671,A -85,B 0,C 180,E1 -13620.353,E2 -13620.353} C_VEL
LIN {X 0,Y 347.698,Z 243.676,A -85,B 0,C 180,E1 -13624.051,E2 -13624.051} C_VEL
LIN {X 0,Y 347.715,Z 243.668,A -85,B 0,C 180,E1 -13627.329,E2 -13627.329} C_VEL
LIN {X 0,Y 347.749,Z 243.67,A -85,B 0,C 180,E1 -13630.297,E2 -13630.297} C_VEL
LIN {X 0,Y 347.778,Z 243.66,A -85,B 0,C 180,E1 -13633.402,E2 -13633.402} C_VEL
LIN {X 0,Y 347.78,Z 243.666,A -85,B 0,C 180,E1 -13636.679,E2 -13636.679} C_VEL
LIN {X 0,Y 347.753,Z 243.665,A -85,B 0,C 180,E1 -13640.174,E2 -13640.174} C_VEL
LIN {X 0,Y 347.761,Z 243.663,A -85,B 0,C 180,E1 -13644.134,E2 -13644.134} C_VEL
LIN {X 0,Y 347.713,Z 243.668,A -85,B 0,C 180,E1 -13648.095,E2 -13648.095} C_VEL
LIN {X 0,Y 347.757,Z 243.669,A -85,B 0,C 180,E1 -13650.997,E2 -13650.997} C_VEL
LIN {X 0,Y 347.811,Z 243.658,A -85,B 0,C 180,E1 -13653.617,E2 -13653.617} C_VEL
LIN {X 0,Y 347.769,Z 243.661,A -85,B 0,C 180,E1 -13656.171,E2 -13656.171} C_VEL
LIN {X 0,Y 347.773,Z 243.662,A -85,B 0,C 180,E1 -13659.917,E2 -13659.917} C_VEL
LIN {X 0,Y 347.824,Z 243.661,A -85,B 0,C 180,E1 -13663.577,E2 -13663.577} C_VEL
LIN {X 0,Y 347.885,Z 243.649,A -85,B 0,C 180,E1 -13667.169,E2 -13667.169} C_VEL
LIN {X 0,Y 347.939,Z 243.64,A -85,B 0,C 180,E1 -13670.709,E2 -13670.709} C_VEL
LIN {X 0,Y 348.044,Z 243.63,A -85,B 0,C 180,E1 -13674.213,E2 -13674.213} C_VEL
LIN {X 0,Y 348.199,Z 243.611,A -85,B 0,C 180,E1 -13677.694,E2 -13677.694} C_VEL
LIN {X 0,Y 348.145,Z 243.615,A -85,B 0,C 180,E1 -13681.164,E2 -13681.164} C_VEL
LIN {X 0,Y 348.195,Z 243.613,A -85,B 0,C 180,E1 -13682.321,E2 -13682.321} C_VEL
LIN {X 0,Y 348.066,Z 243.625,A -85,B 0,C 180,E1 -13686.966,E2 -13686.966} C_VEL
LIN {X 0,Y 347.908,Z 243.65,A -85,B 0,C 180,E1 -13690.482,E2 -13690.482} C_VEL
LIN {X 0,Y 347.916,Z 243.646,A -85,B 0,C 180,E1 -13694.156,E2 -13694.156} C_VEL
LIN {X 0,Y 347.848,Z 243.654,A -85,B 0,C 180,E1 -13698.264,E2 -13698.264} C_VEL
LIN {X 0,Y 347.786,Z 243.659,A -85,B 0,C 180,E1 -13701.631,E2 -13701.631} C_VEL
LIN {X 0,Y 347.787,Z 243.663,A -85,B 0,C 180,E1 -13705.117,E2 -13705.117} C_VEL
LIN {X 0,Y 347.766,Z 243.668,A -85,B 0,C 180,E1 -13709.02,E2 -13709.02} C_VEL
LIN {X 0,Y 347.761,Z 243.663,A -85,B 0,C 180,E1 -13711.917,E2 -13711.917} C_VEL
LIN {X 0,Y 347.811,Z 243.657,A -85,B 0,C 180,E1 -13715.879,E2 -13715.879} C_VEL
LIN {X 0,Y 347.755,Z 243.664,A -85,B 0,C 180,E1 -13718.799,E2 -13718.799} C_VEL
LIN {X 0,Y 347.73,Z 243.669,A -85,B 0,C 180,E1 -13721.84,E2 -13721.84} C_VEL
LIN {X 0,Y 347.711,Z 243.67,A -85,B 0,C 180,E1 -13725.033,E2 -13725.033} C_VEL
LIN {X 0,Y 347.73,Z 243.667,A -85,B 0,C 180,E1 -13728.408,E2 -13728.408} C_VEL
LIN {X 0,Y 347.786,Z 243.664,A -85,B 0,C 180,E1 -13732.016,E2 -13732.016} C_VEL
LIN {X 0,Y 347.768,Z 243.664,A -85,B 0,C 180,E1 -13735.537,E2 -13735.537} C_VEL
LIN {X 0,Y 347.77,Z 243.668,A -85,B 0,C 180,E1 -13738.301,E2 -13738.301} C_VEL
LIN {X 0,Y 347.831,Z 243.805,A -85,B 0,C 180,E1 -13740.88,E2 -13740.88} C_VEL
LIN {X 0,Y 350.249,Z 255.553,A -85,B 0,C 180,E1 -13744.23,E2 -13744.23} C_VEL
LIN {X 0,Y 351.278,Z 262.472,A -85,B 0,C 180,E1 -13746.098,E2 -13746.098} C_VEL
LIN {X 0,Y 350.627,Z 268.761,A -85,B 0,C 180,E1 -13747.639,E2 -13747.639} C_VEL
LIN {X 0,Y 352.597,Z 281.058,A -85,B 0,C 180,E1 -13748.08,E2 -13748.08} C_VEL
LIN {X 0,Y 355.804,Z 301.412,A -85,B 0,C 180,E1 -13748.723,E2 -13748.723} C_VEL
LIN {X 0,Y 354.129,Z 377.02,A -85,B 0,C 180,E1 -13750.394,E2 -13750.394} C_VEL
LIN {X 0,Y 353.488,Z 390.561,A -85,B 0,C 180,E1 -13750.923,E2 -13750.923} C_VEL
LIN {X 0,Y 352.685,Z 402.931,A -85,B 0,C 180,E1 -13751.632,E2 -13751.632} C_VEL
LIN {X 0,Y 351.707,Z 414.84,A -85,B 0,C 180,E1 -13752.556,E2 -13752.556} C_VEL
LIN {X 0,Y 350.665,Z 426.318,A -85,B 0,C 180,E1 -13753.703,E2 -13753.703} C_VEL
LIN {X 0,Y 349.75,Z 436.689,A -85,B 0,C 180,E1 -13755.004,E2 -13755.004} C_VEL
LIN {X 0,Y 348.816,Z 445.152,A -85,B 0,C 180,E1 -13756.304,E2 -13756.304} C_VEL
LIN {X 0,Y 347.834,Z 454.33,A -85,B 0,C 180,E1 -13758.046,E2 -13758.046} C_VEL
LIN {X 0,Y 347.162,Z 461.721,A -85,B 0,C 180,E1 -13759.795,E2 -13759.795} C_VEL
LIN {X 0,Y 346.749,Z 466.706,A -85,B 0,C 180,E1 -13761.255,E2 -13761.255} C_VEL
LIN {X 0,Y 346.393,Z 471.531,A -85,B 0,C 180,E1 -13763.006,E2 -13763.006} C_VEL
LIN {X 0,Y 346.201,Z 474.774,A -85,B 0,C 180,E1 -13764.523,E2 -13764.523} C_VEL
LIN {X 0,Y 346.134,Z 477.839,A -85,B 0,C 180,E1 -13766.506,E2 -13766.506} C_VEL
LIN {X 0,Y 346.059,Z 479.07,A -85,B 0,C 180,E1 -13767.67,E2 -13767.67} C_VEL
LIN {X 0,Y 346.061,Z 479.856,A -85,B 0,C 180,E1 -13768.834,E2 -13768.834} C_VEL
LIN {X 0,Y 346.087,Z 480.224,A -85,B 0,C 180,E1 -13769.998,E2 -13769.998} C_VEL
LIN {X 0,Y 346.06,Z 480.197,A -85,B 0,C 180,E1 -13771.162,E2 -13771.162} C_VEL
LIN {X 0,Y 346.057,Z 479.778,A -85,B 0,C 180,E1 -13772.326,E2 -13772.326} C_VEL
LIN {X 0,Y 346.135,Z 478.92,A -85,B 0,C 180,E1 -13773.49,E2 -13773.49} C_VEL
LIN {X 0,Y 346.188,Z 477.645,A -85,B 0,C 180,E1 -13774.656,E2 -13774.656} C_VEL
LIN {X 0,Y 346.299,Z 475.662,A -85,B 0,C 180,E1 -13776.012,E2 -13776.012} C_VEL
LIN {X 0,Y 346.674,Z 471.221,A -85,B 0,C 180,E1 -13778.156,E2 -13778.156} C_VEL
LIN {X 0,Y 347.205,Z 466.371,A -85,B 0,C 180,E1 -13779.905,E2 -13779.905} C_VEL
LIN {X 0,Y 347.946,Z 460.254,A -85,B 0,C 180,E1 -13781.651,E2 -13781.651} C_VEL
LIN {X 0,Y 349.013,Z 452.653,A -85,B 0,C 180,E1 -13783.387,E2 -13783.387} C_VEL
LIN {X 0,Y 350.134,Z 444.903,A -85,B 0,C 180,E1 -13784.826,E2 -13784.826} C_VEL
LIN {X 0,Y 351.351,Z 434.426,A -85,B 0,C 180,E1 -13786.41,E2 -13786.41} C_VEL
LIN {X 0,Y 352.642,Z 423.806,A -85,B 0,C 180,E1 -13787.691,E2 -13787.691} C_VEL
LIN {X 0,Y 354.011,Z 411.916,A -85,B 0,C 180,E1 -13788.818,E2 -13788.818} C_VEL
LIN {X 0,Y 355.158,Z 400.395,A -85,B 0,C 180,E1 -13789.655,E2 -13789.655} C_VEL
LIN {X 0,Y 356.104,Z 386.804,A -85,B 0,C 180,E1 -13790.391,E2 -13790.391} C_VEL
LIN {X 0,Y 356.798,Z 374.05,A -85,B 0,C 180,E1 -13790.832,E2 -13790.832} C_VEL
LIN {X 0,Y 358.614,Z 302.005,A -85,B 0,C 180,E1 -13792.454,E2 -13792.454} C_VEL
LIN {X 0,Y 355.641,Z 284.221,A -85,B 0,C 180,E1 -13793.135,E2 -13793.135} C_VEL
LIN {X 0,Y 352.091,Z 267.722,A -85,B 0,C 180,E1 -13793.892,E2 -13793.892} C_VEL
LIN {X 0,Y 352.146,Z 264.154,A -85,B 0,C 180,E1 -13794.776,E2 -13794.776} C_VEL
LIN {X 0,Y 350.363,Z 254.451,A -85,B 0,C 180,E1 -13797.472,E2 -13797.472} C_VEL
LIN {X 0,Y 347.82,Z 243.838,A -85,B 0,C 180,E1 -13800.674,E2 -13800.674} C_VEL
LIN {X 0,Y 347.756,Z 243.667,A -85,B 0,C 180,E1 -13804.46,E2 -13804.46} C_VEL
LIN {X 0,Y 347.772,Z 243.666,A -85,B 0,C 180,E1 -13807.981,E2 -13807.981} C_VEL
LIN {X 0,Y 347.748,Z 243.668,A -85,B 0,C 180,E1 -13811.827,E2 -13811.827} C_VEL
LIN {X 0,Y 347.706,Z 243.671,A -85,B 0,C 180,E1 -13815.023,E2 -13815.023} C_VEL
LIN {X 0,Y 347.744,Z 243.667,A -85,B 0,C 180,E1 -13818.394,E2 -13818.394} C_VEL
LIN {X 0,Y 347.766,Z 243.666,A -85,B 0,C 180,E1 -13822.009,E2 -13822.009} C_VEL
LIN {X 0,Y 347.746,Z 243.667,A -85,B 0,C 180,E1 -13825.53,E2 -13825.53} C_VEL
LIN {X 0,Y 347.747,Z 243.668,A -85,B 0,C 180,E1 -13828.294,E2 -13828.294} C_VEL
LIN {X 0,Y 347.743,Z 243.667,A -85,B 0,C 180,E1 -13830.978,E2 -13830.978} C_VEL
LIN {X 0,Y 347.762,Z 243.666,A -85,B 0,C 180,E1 -13834.881,E2 -13834.881} C_VEL
LIN {X 0,Y 347.775,Z 243.664,A -85,B 0,C 180,E1 -13838.663,E2 -13838.663} C_VEL
LIN {X 0,Y 347.793,Z 243.661,A -85,B 0,C 180,E1 -13842.349,E2 -13842.349} C_VEL
LIN {X 0,Y 347.892,Z 243.649,A -85,B 0,C 180,E1 -13845.964,E2 -13845.964} C_VEL
LIN {X 0,Y 347.884,Z 243.651,A -85,B 0,C 180,E1 -13849.517,E2 -13849.517} C_VEL
LIN {X 0,Y 348.056,Z 243.632,A -85,B 0,C 180,E1 -13853.034,E2 -13853.034} C_VEL
LIN {X 0,Y 348.175,Z 243.612,A -85,B 0,C 180,E1 -13857.679,E2 -13857.679} C_VEL
LIN {X 0,Y 348.287,Z 243.596,A -85,B 0,C 180,E1 -13859.992,E2 -13859.992} C_VEL
LIN {X 0,Y 348.187,Z 243.61,A -85,B 0,C 180,E1 -13862.306,E2 -13862.306} C_VEL
LIN {X 0,Y 348.058,Z 243.629,A -85,B 0,C 180,E1 -13866.95,E2 -13866.95} C_VEL
LIN {X 0,Y 347.941,Z 243.644,A -85,B 0,C 180,E1 -13869.291,E2 -13869.291} C_VEL
LIN {X 0,Y 347.867,Z 243.654,A -85,B 0,C 180,E1 -13872.832,E2 -13872.832} C_VEL
LIN {X 0,Y 347.812,Z 243.662,A -85,B 0,C 180,E1 -13876.424,E2 -13876.424} C_VEL
LIN {X 0,Y 347.849,Z 243.701,A -85,B 0,C 180,E1 -13877.632,E2 -13877.632} C_VEL
LIN {X 0,Y 348.727,Z 247.403,A -85,B 0,C 180,E1 -13878.802,E2 -13878.802} C_VEL
LIN {X 0,Y 351.064,Z 257.825,A -85,B 0,C 180,E1 -13881.728,E2 -13881.728} C_VEL
LIN {X 0,Y 351.464,Z 259.553,A -85,B 0,C 180,E1 -13882.126,E2 -13882.126} C_VEL
LIN {X 0,Y 354.335,Z 266.879,A -85,B 0,C 180,E1 -13882.569,E2 -13882.569} C_VEL
LIN {X 0,Y 358.466,Z 286.983,A -85,B 0,C 180,E1 -13883.42,E2 -13883.42} C_VEL
LIN {X 0,Y 358.855,Z 290.889,A -85,B 0,C 180,E1 -13883.546,E2 -13883.546} C_VEL
LIN {X 0,Y 356.777,Z 368.048,A -85,B 0,C 180,E1 -13885.297,E2 -13885.297} C_VEL
LIN {X 0,Y 356.033,Z 381.846,A -85,B 0,C 180,E1 -13885.847,E2 -13885.847} C_VEL
LIN {X 0,Y 355.106,Z 394.472,A -85,B 0,C 180,E1 -13886.591,E2 -13886.591} C_VEL
LIN {X 0,Y 353.957,Z 406.651,A -85,B 0,C 180,E1 -13887.563,E2 -13887.563} C_VEL
LIN {X 0,Y 352.651,Z 418.138,A -85,B 0,C 180,E1 -13888.738,E2 -13888.738} C_VEL
LIN {X 0,Y 351.418,Z 427.861,A -85,B 0,C 180,E1 -13889.987,E2 -13889.987} C_VEL
LIN {X 0,Y 350.205,Z 437.024,A -85,B 0,C 180,E1 -13891.44,E2 -13891.44} C_VEL
LIN {X 0,Y 348.897,Z 446.193,A -85,B 0,C 180,E1 -13893.237,E2 -13893.237} C_VEL
LIN {X 0,Y 347.918,Z 453.762,A -85,B 0,C 180,E1 -13895.137,E2 -13895.137} C_VEL
LIN {X 0,Y 347.166,Z 459.661,A -85,B 0,C 180,E1 -13897.027,E2 -13897.027} C_VEL
LIN {X 0,Y 346.599,Z 464.213,A -85,B 0,C 180,E1 -13898.933,E2 -13898.933} C_VEL
LIN {X 0,Y 346.15,Z 468.102,A -85,B 0,C 180,E1 -13901.307,E2 -13901.307} C_VEL
LIN {X 0,Y 345.938,Z 470.251,A -85,B 0,C 180,E1 -13903.674,E2 -13903.674} C_VEL
LIN {X 0,Y 345.851,Z 470.72,A -85,B 0,C 180,E1 -13905.32,E2 -13905.32} C_VEL
LIN {X 0,Y 345.829,Z 470.364,A -85,B 0,C 180,E1 -13907.005,E2 -13907.005} C_VEL
LIN {X 0,Y 345.89,Z 469.122,A -85,B 0,C 180,E1 -13908.729,E2 -13908.729} C_VEL
LIN {X 0,Y 346.161,Z 466.108,A -85,B 0,C 180,E1 -13910.999,E2 -13910.999} C_VEL
LIN {X 0,Y 346.513,Z 461.359,A -85,B 0,C 180,E1 -13913.253,E2 -13913.253} C_VEL
LIN {X 0,Y 347.015,Z 455.951,A -85,B 0,C 180,E1 -13915.14,E2 -13915.14} C_VEL
LIN {X 0,Y 347.639,Z 449.433,A -85,B 0,C 180,E1 -13916.921,E2 -13916.921} C_VEL
LIN {X 0,Y 348.45,Z 441.131,A -85,B 0,C 180,E1 -13918.713,E2 -13918.713} C_VEL
LIN {X 0,Y 349.349,Z 432.581,A -85,B 0,C 180,E1 -13920.207,E2 -13920.207} C_VEL
LIN {X 0,Y 350.303,Z 422.944,A -85,B 0,C 180,E1 -13921.584,E2 -13921.584} C_VEL
LIN {X 0,Y 351.279,Z 412.711,A -85,B 0,C 180,E1 -13922.762,E2 -13922.762} C_VEL
LIN {X 0,Y 352.284,Z 400.919,A -85,B 0,C 180,E1 -13923.838,E2 -13923.838} C_VEL
LIN {X 0,Y 353.068,Z 389.227,A -85,B 0,C 180,E1 -13924.664,E2 -13924.664} C_VEL
LIN {X 0,Y 353.791,Z 376.716,A -85,B 0,C 180,E1 -13925.308,E2 -13925.308} C_VEL
LIN {X 0,Y 354.274,Z 363.658,A -85,B 0,C 180,E1 -13925.745,E2 -13925.745} C_VEL
LIN {X 0,Y 355.823,Z 287.866,A -85,B 0,C 180,E1 -13927.406,E2 -13927.406} C_VEL
LIN {X 0,Y 350.867,Z 260.593,A -85,B 0,C 180,E1 -13928.329,E2 -13928.329} C_VEL
LIN {X 0,Y 350.714,Z 259.332,A -85,B 0,C 180,E1 -13928.474,E2 -13928.474} C_VEL
LIN {X 0,Y 349.029,Z 249.889,A -85,B 0,C 180,E1 -13931.208,E2 -13931.208} C_VEL
LIN {X 0,Y 347.82,Z 243.719,A -85,B 0,C 180,E1 -13933.117,E2 -13933.117} C_VEL
LIN {X 0,Y 347.822,Z 243.656,A -85,B 0,C 180,E1 -13937.16,E2 -13937.16} C_VEL
LIN {X 0,Y 347.894,Z 243.653,A -85,B 0,C 180,E1 -13940.702,E2 -13940.702} C_VEL
LIN {X 0,Y 348.024,Z 243.633,A -85,B 0,C 180,E1 -13943.043,E2 -13943.043} C_VEL
LIN {X 0,Y 348.145,Z 243.615,A -85,B 0,C 180,E1 -13947.688,E2 -13947.688} C_VEL
LIN {X 0,Y 348.277,Z 243.598,A -85,B 0,C 180,E1 -13950.002,E2 -13950.002} C_VEL
LIN {X 0,Y 348.146,Z 243.615,A -85,B 0,C 180,E1 -13952.316,E2 -13952.316} C_VEL
LIN {X 0,Y 348.027,Z 243.633,A -85,B 0,C 180,E1 -13956.961,E2 -13956.961} C_VEL
LIN {X 0,Y 347.866,Z 243.649,A -85,B 0,C 180,E1 -13960.478,E2 -13960.478} C_VEL
LIN {X 0,Y 347.834,Z 243.654,A -85,B 0,C 180,E1 -13964.154,E2 -13964.154} C_VEL
LIN {X 0,Y 347.821,Z 243.656,A -85,B 0,C 180,E1 -13968.201,E2 -13968.201} C_VEL
LIN {X 0,Y 347.192,Z 243.737,A -85,B 0,C 180,E1 -13969.166,E2 -13969.166} C_VEL
LIN {X 0,Y 344.303,Z 244.094,A -85,B 0,C 180,E1 -13970.735,E2 -13970.735} C_VEL
LIN {X 0,Y 341.822,Z 244.406,A -85,B 0,C 180,E1 -13972.005,E2 -13972.005} C_VEL
LIN {X 0,Y 340.749,Z 244.536,A -85,B 0,C 180,E1 -13972.99,E2 -13972.99} C_VEL
LIN {X 0,Y 340.66,Z 244.546,A -85,B 0,C 180,E1 -13973.323,E2 -13973.323} C_VEL
LIN {X 0,Y 340.748,Z 244.536,A -85,B 0,C 180,E1 -13976.987,E2 -13976.987} C_VEL
LIN {X 0,Y 340.712,Z 244.547,A -85,B 0,C 180,E1 -13979.985,E2 -13979.985} C_VEL
LIN {X 0,Y 340.645,Z 244.552,A -85,B 0,C 180,E1 -13983.854,E2 -13983.854} C_VEL
LIN {X 0,Y 340.657,Z 244.549,A -85,B 0,C 180,E1 -13986.749,E2 -13986.749} C_VEL
LIN {X 0,Y 340.72,Z 244.545,A -85,B 0,C 180,E1 -13990.27,E2 -13990.27} C_VEL
LIN {X 0,Y 340.738,Z 244.538,A -85,B 0,C 180,E1 -13993.804,E2 -13993.804} C_VEL
LIN {X 0,Y 340.724,Z 244.54,A -85,B 0,C 180,E1 -13997.118,E2 -13997.118} C_VEL
LIN {X 0,Y 340.702,Z 244.544,A -85,B 0,C 180,E1 -14000.261,E2 -14000.261} C_VEL
LIN {X 0,Y 340.683,Z 244.544,A -85,B 0,C 180,E1 -14003.568,E2 -14003.568} C_VEL
LIN {X 0,Y 340.665,Z 244.547,A -85,B 0,C 180,E1 -14006.162,E2 -14006.162} C_VEL
LIN {X 0,Y 340.719,Z 244.54,A -85,B 0,C 180,E1 -14010.338,E2 -14010.338} C_VEL
LIN {X 0,Y 340.772,Z 244.538,A -85,B 0,C 180,E1 -14013.028,E2 -14013.028} C_VEL
LIN {X 0,Y 340.738,Z 244.54,A -85,B 0,C 180,E1 -14015.647,E2 -14015.647} C_VEL
LIN {X 0,Y 340.709,Z 244.546,A -85,B 0,C 180,E1 -14019.482,E2 -14019.482} C_VEL
LIN {X 0,Y 340.782,Z 244.533,A -85,B 0,C 180,E1 -14021.99,E2 -14021.99} C_VEL
LIN {X 0,Y 340.864,Z 244.527,A -85,B 0,C 180,E1 -14025.714,E2 -14025.714} C_VEL
LIN {X 0,Y 340.867,Z 244.524,A -85,B 0,C 180,E1 -14029.315,E2 -14029.315} C_VEL
LIN {X 0,Y 341.003,Z 244.504,A -85,B 0,C 180,E1 -14032.905,E2 -14032.905} C_VEL
LIN {X 0,Y 340.827,Z 244.527,A -85,B 0,C 180,E1 -14035.277,E2 -14035.277} C_VEL
LIN {X 0,Y 341.137,Z 244.491,A -85,B 0,C 180,E1 -14037.646,E2 -14037.646} C_VEL
LIN {X 0,Y 341.114,Z 244.49,A -85,B 0,C 180,E1 -14041.188,E2 -14041.188} C_VEL
LIN {X 0,Y 341.132,Z 244.492,A -85,B 0,C 180,E1 -14042.369,E2 -14042.369} C_VEL
LIN {X 0,Y 341.025,Z 244.504,A -85,B 0,C 180,E1 -14045.922,E2 -14045.922} C_VEL
LIN {X 0,Y 340.977,Z 244.514,A -85,B 0,C 180,E1 -14048.363,E2 -14048.363} C_VEL
LIN {X 0,Y 340.863,Z 244.523,A -85,B 0,C 180,E1 -14051.906,E2 -14051.906} C_VEL
LIN {X 0,Y 340.834,Z 244.525,A -85,B 0,C 180,E1 -14055.556,E2 -14055.556} C_VEL
LIN {X 0,Y 340.746,Z 244.537,A -85,B 0,C 180,E1 -14059.276,E2 -14059.276} C_VEL
LIN {X 0,Y 340.73,Z 244.542,A -85,B 0,C 180,E1 -14063.079,E2 -14063.079} C_VEL
LIN {X 0,Y 340.736,Z 244.538,A -85,B 0,C 180,E1 -14065.674,E2 -14065.674} C_VEL
LIN {X 0,Y 340.725,Z 244.54,A -85,B 0,C 180,E1 -14069.679,E2 -14069.679} C_VEL
LIN {X 0,Y 340.71,Z 244.541,A -85,B 0,C 180,E1 -14072.44,E2 -14072.44} C_VEL
LIN {X 0,Y 340.741,Z 244.543,A -85,B 0,C 180,E1 -14075.283,E2 -14075.283} C_VEL
LIN {X 0,Y 340.718,Z 244.54,A -85,B 0,C 180,E1 -14078.385,E2 -14078.385} C_VEL
LIN {X 0,Y 340.687,Z 244.545,A -85,B 0,C 180,E1 -14082.041,E2 -14082.041} C_VEL
LIN {X 0,Y 340.651,Z 244.553,A -85,B 0,C 180,E1 -14085.454,E2 -14085.454} C_VEL
LIN {X 0,Y 340.668,Z 244.546,A -85,B 0,C 180,E1 -14088.686,E2 -14088.686} C_VEL
LIN {X 0,Y 340.743,Z 244.543,A -85,B 0,C 180,E1 -14091.772,E2 -14091.772} C_VEL
LIN {X 0,Y 340.747,Z 244.539,A -85,B 0,C 180,E1 -14095.597,E2 -14095.597} C_VEL
LIN {X 0,Y 340.717,Z 244.543,A -85,B 0,C 180,E1 -14098.955,E2 -14098.955} C_VEL
LIN {X 0,Y 340.768,Z 244.699,A -85,B 0,C 180,E1 -14100.585,E2 -14100.585} C_VEL
LIN {X 0,Y 343.37,Z 257.304,A -85,B 0,C 180,E1 -14104.244,E2 -14104.244} C_VEL
LIN {X 0,Y 344.322,Z 263.315,A -85,B 0,C 180,E1 -14105.905,E2 -14105.905} C_VEL
LIN {X 0,Y 343.75,Z 268.679,A -85,B 0,C 180,E1 -14107.236,E2 -14107.236} C_VEL
LIN {X 0,Y 344.979,Z 276.327,A -85,B 0,C 180,E1 -14107.54,E2 -14107.54} C_VEL
LIN {X 0,Y 349.031,Z 302.238,A -85,B 0,C 180,E1 -14108.384,E2 -14108.384} C_VEL
LIN {X 0,Y 347.321,Z 376.952,A -85,B 0,C 180,E1 -14110.071,E2 -14110.071} C_VEL
LIN {X 0,Y 346.667,Z 390.475,A -85,B 0,C 180,E1 -14110.61,E2 -14110.61} C_VEL
LIN {X 0,Y 345.833,Z 402.836,A -85,B 0,C 180,E1 -14111.331,E2 -14111.331} C_VEL
LIN {X 0,Y 344.893,Z 413.949,A -85,B 0,C 180,E1 -14112.2,E2 -14112.2} C_VEL
LIN {X 0,Y 343.789,Z 425.568,A -85,B 0,C 180,E1 -14113.368,E2 -14113.368} C_VEL
LIN {X 0,Y 342.879,Z 435.525,A -85,B 0,C 180,E1 -14114.621,E2 -14114.621} C_VEL
LIN {X 0,Y 341.852,Z 444.629,A -85,B 0,C 180,E1 -14116.019,E2 -14116.019} C_VEL
LIN {X 0,Y 341.034,Z 452.52,A -85,B 0,C 180,E1 -14117.501,E2 -14117.501} C_VEL
LIN {X 0,Y 340.251,Z 460.212,A -85,B 0,C 180,E1 -14119.285,E2 -14119.285} C_VEL
LIN {X 0,Y 339.713,Z 466.388,A -85,B 0,C 180,E1 -14121.072,E2 -14121.072} C_VEL
LIN {X 0,Y 339.314,Z 471.261,A -85,B 0,C 180,E1 -14122.859,E2 -14122.859} C_VEL
LIN {X 0,Y 339.096,Z 474.905,A -85,B 0,C 180,E1 -14124.604,E2 -14124.604} C_VEL
LIN {X 0,Y 339.06,Z 477.656,A -85,B 0,C 180,E1 -14126.433,E2 -14126.433} C_VEL
LIN {X 0,Y 338.976,Z 478.907,A -85,B 0,C 180,E1 -14127.621,E2 -14127.621} C_VEL
LIN {X 0,Y 338.967,Z 479.729,A -85,B 0,C 180,E1 -14128.81,E2 -14128.81} C_VEL
LIN {X 0,Y 338.99,Z 480.115,A -85,B 0,C 180,E1 -14129.998,E2 -14129.998} C_VEL
LIN {X 0,Y 338.966,Z 480.106,A -85,B 0,C 180,E1 -14131.186,E2 -14131.186} C_VEL
LIN {X 0,Y 338.975,Z 479.704,A -85,B 0,C 180,E1 -14132.374,E2 -14132.374} C_VEL
LIN {X 0,Y 339.063,Z 478.88,A -85,B 0,C 180,E1 -14133.563,E2 -14133.563} C_VEL
LIN {X 0,Y 339.094,Z 477.621,A -85,B 0,C 180,E1 -14134.753,E2 -14134.753} C_VEL
LIN {X 0,Y 339.272,Z 474.956,A -85,B 0,C 180,E1 -14136.54,E2 -14136.54} C_VEL
LIN {X 0,Y 339.624,Z 471.263,A -85,B 0,C 180,E1 -14138.327,E2 -14138.327} C_VEL
LIN {X 0,Y 340.186,Z 466.448,A -85,B 0,C 180,E1 -14140.112,E2 -14140.112} C_VEL
LIN {X 0,Y 340.967,Z 460.378,A -85,B 0,C 180,E1 -14141.893,E2 -14141.893} C_VEL
LIN {X 0,Y 342.117,Z 452.842,A -85,B 0,C 180,E1 -14143.662,E2 -14143.662} C_VEL
LIN {X 0,Y 343.274,Z 445.168,A -85,B 0,C 180,E1 -14145.129,E2 -14145.129} C_VEL
LIN {X 0,Y 344.431,Z 435.883,A -85,B 0,C 180,E1 -14146.596,E2 -14146.596} C_VEL
LIN {X 0,Y 345.762,Z 425.577,A -85,B 0,C 180,E1 -14147.902,E2 -14147.902} C_VEL
LIN {X 0,Y 347.188,Z 414.192,A -85,B 0,C 180,E1 -14149.049,E2 -14149.049} C_VEL
LIN {X 0,Y 348.38,Z 402.406,A -85,B 0,C 180,E1 -14149.977,E2 -14149.977} C_VEL
LIN {X 0,Y 349.395,Z 389.529,A -85,B 0,C 180,E1 -14150.723,E2 -14150.723} C_VEL
LIN {X 0,Y 350.222,Z 376.197,A -85,B 0,C 180,E1 -14151.245,E2 -14151.245} C_VEL
LIN {X 0,Y 352.249,Z 303.032,A -85,B 0,C 180,E1 -14152.936,E2 -14152.936} C_VEL
LIN {X 0,Y 349.181,Z 284.5,A -85,B 0,C 180,E1 -14153.675,E2 -14153.675} C_VEL
LIN {X 0,Y 345.439,Z 267.665,A -85,B 0,C 180,E1 -14154.48,E2 -14154.48} C_VEL
LIN {X 0,Y 344.573,Z 261.424,A -85,B 0,C 180,E1 -14156.168,E2 -14156.168} C_VEL
LIN {X 0,Y 342.66,Z 252.449,A -85,B 0,C 180,E1 -14158.812,E2 -14158.812} C_VEL
LIN {X 0,Y 340.747,Z 244.648,A -85,B 0,C 180,E1 -14161.296,E2 -14161.296} C_VEL
LIN {X 0,Y 340.729,Z 244.544,A -85,B 0,C 180,E1 -14165.275,E2 -14165.275} C_VEL
LIN {X 0,Y 340.704,Z 244.547,A -85,B 0,C 180,E1 -14168.377,E2 -14168.377} C_VEL
LIN {X 0,Y 340.699,Z 244.548,A -85,B 0,C 180,E1 -14172.038,E2 -14172.038} C_VEL
LIN {X 0,Y 340.656,Z 244.551,A -85,B 0,C 180,E1 -14176.222,E2 -14176.222} C_VEL
LIN {X 0,Y 340.675,Z 244.549,A -85,B 0,C 180,E1 -14178.682,E2 -14178.682} C_VEL
LIN {X 0,Y 340.723,Z 244.541,A -85,B 0,C 180,E1 -14181.765,E2 -14181.765} C_VEL
LIN {X 0,Y 340.726,Z 244.542,A -85,B 0,C 180,E1 -14185.59,E2 -14185.59} C_VEL
LIN {X 0,Y 340.696,Z 244.545,A -85,B 0,C 180,E1 -14188.948,E2 -14188.948} C_VEL
LIN {X 0,Y 340.711,Z 244.538,A -85,B 0,C 180,E1 -14193.005,E2 -14193.005} C_VEL
LIN {X 0,Y 340.743,Z 244.539,A -85,B 0,C 180,E1 -14195.631,E2 -14195.631} C_VEL
LIN {X 0,Y 340.703,Z 244.544,A -85,B 0,C 180,E1 -14199.465,E2 -14199.465} C_VEL
LIN {X 0,Y 340.747,Z 244.537,A -85,B 0,C 180,E1 -14201.971,E2 -14201.971} C_VEL
LIN {X 0,Y 340.826,Z 244.529,A -85,B 0,C 180,E1 -14205.723,E2 -14205.723} C_VEL
LIN {X 0,Y 340.836,Z 244.531,A -85,B 0,C 180,E1 -14209.298,E2 -14209.298} C_VEL
LIN {X 0,Y 341.001,Z 244.51,A -85,B 0,C 180,E1 -14212.889,E2 -14212.889} C_VEL
LIN {X 0,Y 340.806,Z 244.532,A -85,B 0,C 180,E1 -14215.261,E2 -14215.261} C_VEL
LIN {X 0,Y 341.112,Z 244.492,A -85,B 0,C 180,E1 -14217.631,E2 -14217.631} C_VEL
LIN {X 0,Y 341.238,Z 244.474,A -85,B 0,C 180,E1 -14219.992,E2 -14219.992} C_VEL
LIN {X 0,Y 341.149,Z 244.486,A -85,B 0,C 180,E1 -14222.353,E2 -14222.353} C_VEL
LIN {X 0,Y 341.028,Z 244.504,A -85,B 0,C 180,E1 -14227.094,E2 -14227.094} C_VEL
LIN {X 0,Y 340.85,Z 244.526,A -85,B 0,C 180,E1 -14230.686,E2 -14230.686} C_VEL
LIN {X 0,Y 340.835,Z 244.531,A -85,B 0,C 180,E1 -14234.317,E2 -14234.317} C_VEL
LIN {X 0,Y 340.836,Z 244.73,A -85,B 0,C 180,E1 -14237.155,E2 -14237.155} C_VEL
LIN {X 0,Y 343.398,Z 255.386,A -85,B 0,C 180,E1 -14240.351,E2 -14240.351} C_VEL
LIN {X 0,Y 344.29,Z 259.579,A -85,B 0,C 180,E1 -14241.469,E2 -14241.469} C_VEL
LIN {X 0,Y 348.352,Z 269.601,A -85,B 0,C 180,E1 -14242.12,E2 -14242.12} C_VEL
LIN {X 0,Y 352.45,Z 289.885,A -85,B 0,C 180,E1 -14243.001,E2 -14243.001} C_VEL
LIN {X 0,Y 350.299,Z 368.279,A -85,B 0,C 180,E1 -14244.829,E2 -14244.829} C_VEL
LIN {X 0,Y 349.536,Z 381.966,A -85,B 0,C 180,E1 -14245.385,E2 -14245.385} C_VEL
LIN {X 0,Y 348.641,Z 393.884,A -85,B 0,C 180,E1 -14246.093,E2 -14246.093} C_VEL
LIN {X 0,Y 347.52,Z 405.226,A -85,B 0,C 180,E1 -14246.988,E2 -14246.988} C_VEL
LIN {X 0,Y 346.152,Z 416.772,A -85,B 0,C 180,E1 -14248.157,E2 -14248.157} C_VEL
LIN {X 0,Y 344.843,Z 426.878,A -85,B 0,C 180,E1 -14249.44,E2 -14249.44} C_VEL
LIN {X 0,Y 343.643,Z 435.625,A -85,B 0,C 180,E1 -14250.805,E2 -14250.805} C_VEL
LIN {X 0,Y 342.534,Z 443.152,A -85,B 0,C 180,E1 -14252.228,E2 -14252.228} C_VEL
LIN {X 0,Y 341.346,Z 451.227,A -85,B 0,C 180,E1 -14254.122,E2 -14254.122} C_VEL
LIN {X 0,Y 340.51,Z 456.986,A -85,B 0,C 180,E1 -14255.81,E2 -14255.81} C_VEL
LIN {X 0,Y 339.914,Z 461.571,A -85,B 0,C 180,E1 -14257.489,E2 -14257.489} C_VEL
LIN {X 0,Y 339.475,Z 465.113,A -85,B 0,C 180,E1 -14259.142,E2 -14259.142} C_VEL
LIN {X 0,Y 339.139,Z 467.699,A -85,B 0,C 180,E1 -14260.737,E2 -14260.737} C_VEL
LIN {X 0,Y 339.018,Z 468.9,A -85,B 0,C 180,E1 -14261.733,E2 -14261.733} C_VEL
LIN {X 0,Y 338.864,Z 470.294,A -85,B 0,C 180,E1 -14263.46,E2 -14263.46} C_VEL
LIN {X 0,Y 338.771,Z 470.808,A -85,B 0,C 180,E1 -14265.146,E2 -14265.146} C_VEL
LIN {X 0,Y 338.725,Z 470.535,A -85,B 0,C 180,E1 -14266.792,E2 -14266.792} C_VEL
LIN {X 0,Y 338.793,Z 469.519,A -85,B 0,C 180,E1 -14268.412,E2 -14268.412} C_VEL
LIN {X 0,Y 338.948,Z 467.65,A -85,B 0,C 180,E1 -14270.085,E2 -14270.085} C_VEL
LIN {X 0,Y 339.201,Z 464.599,A -85,B 0,C 180,E1 -14271.919,E2 -14271.919} C_VEL
LIN {X 0,Y 339.575,Z 460.297,A -85,B 0,C 180,E1 -14273.801,E2 -14273.801} C_VEL
LIN {X 0,Y 340.1,Z 454.49,A -85,B 0,C 180,E1 -14275.729,E2 -14275.729} C_VEL
LIN {X 0,Y 340.847,Z 446.936,A -85,B 0,C 180,E1 -14277.693,E2 -14277.693} C_VEL
LIN {X 0,Y 341.732,Z 438.626,A -85,B 0,C 180,E1 -14279.404,E2 -14279.404} C_VEL
LIN {X 0,Y 342.701,Z 429.207,A -85,B 0,C 180,E1 -14280.966,E2 -14280.966} C_VEL
LIN {X 0,Y 343.875,Z 417.952,A -85,B 0,C 180,E1 -14282.461,E2 -14282.461} C_VEL
LIN {X 0,Y 344.94,Z 406.26,A -85,B 0,C 180,E1 -14283.674,E2 -14283.674} C_VEL
LIN {X 0,Y 345.95,Z 393.901,A -85,B 0,C 180,E1 -14284.669,E2 -14284.669} C_VEL
LIN {X 0,Y 346.707,Z 381.314,A -85,B 0,C 180,E1 -14285.415,E2 -14285.415} C_VEL
LIN {X 0,Y 347.371,Z 367.403,A -85,B 0,C 180,E1 -14285.971,E2 -14285.971} C_VEL
LIN {X 0,Y 349.073,Z 288.917,A -85,B 0,C 180,E1 -14287.746,E2 -14287.746} C_VEL
LIN {X 0,Y 344.131,Z 261.732,A -85,B 0,C 180,E1 -14288.67,E2 -14288.67} C_VEL
LIN {X 0,Y 343.607,Z 259.639,A -85,B 0,C 180,E1 -14288.833,E2 -14288.833} C_VEL
LIN {X 0,Y 341.614,Z 248.889,A -85,B 0,C 180,E1 -14292.028,E2 -14292.028} C_VEL
LIN {X 0,Y 340.769,Z 244.589,A -85,B 0,C 180,E1 -14293.413,E2 -14293.413} C_VEL
LIN {X 0,Y 340.776,Z 244.536,A -85,B 0,C 180,E1 -14296.89,E2 -14296.89} C_VEL
LIN {X 0,Y 340.857,Z 244.527,A -85,B 0,C 180,E1 -14300.508,E2 -14300.508} C_VEL
LIN {X 0,Y 340.992,Z 244.511,A -85,B 0,C 180,E1 -14302.899,E2 -14302.899} C_VEL
LIN {X 0,Y 341.108,Z 244.492,A -85,B 0,C 180,E1 -14307.64,E2 -14307.64} C_VEL
LIN {X 0,Y 341.227,Z 244.476,A -85,B 0,C 180,E1 -14310.002,E2 -14310.002} C_VEL
LIN {X 0,Y 341.109,Z 244.492,A -85,B 0,C 180,E1 -14312.364,E2 -14312.364} C_VEL
LIN {X 0,Y 340.995,Z 244.51,A -85,B 0,C 180,E1 -14317.105,E2 -14317.105} C_VEL
LIN {X 0,Y 340.808,Z 244.529,A -85,B 0,C 180,E1 -14320.698,E2 -14320.698} C_VEL
LIN {X 0,Y 340.799,Z 244.53,A -85,B 0,C 180,E1 -14324.329,E2 -14324.329} C_VEL
LIN {X 0,Y 340.774,Z 244.533,A -85,B 0,C 180,E1 -14328.471,E2 -14328.471} C_VEL
LIN {X 0,Y 340.662,Z 244.552,A -85,B 0,C 180,E1 -14331.849,E2 -14331.849} C_VEL
LIN {X 0,Y 340.66,Z 244.546,A -85,B 0,C 180,E1 -14333.323,E2 -14333.323} C_VEL
LIN {X 0,Y 339.988,Z 244.633,A -85,B 0,C 180,E1 -14334.31,E2 -14334.31} C_VEL
LIN {X 0,Y 337.143,Z 244.991,A -85,B 0,C 180,E1 -14335.916,E2 -14335.916} C_VEL
LIN {X 0,Y 334.743,Z 245.288,A -85,B 0,C 180,E1 -14337.216,E2 -14337.216} C_VEL
LIN {X 0,Y 333.723,Z 245.413,A -85,B 0,C 180,E1 -14338.223,E2 -14338.223} C_VEL
LIN {X 0,Y 333.645,Z 245.419,A -85,B 0,C 180,E1 -14338.563,E2 -14338.563} C_VEL
LIN {X 0,Y 333.591,Z 245.43,A -85,B 0,C 180,E1 -14341.784,E2 -14341.784} C_VEL
LIN {X 0,Y 333.636,Z 245.423,A -85,B 0,C 180,E1 -14344.781,E2 -14344.781} C_VEL
LIN {X 0,Y 333.634,Z 245.424,A -85,B 0,C 180,E1 -14348.812,E2 -14348.812} C_VEL
LIN {X 0,Y 333.662,Z 245.425,A -85,B 0,C 180,E1 -14352.522,E2 -14352.522} C_VEL
LIN {X 0,Y 333.691,Z 245.416,A -85,B 0,C 180,E1 -14355.986,E2 -14355.986} C_VEL
LIN {X 0,Y 333.668,Z 245.419,A -85,B 0,C 180,E1 -14359.313,E2 -14359.313} C_VEL
LIN {X 0,Y 333.638,Z 245.424,A -85,B 0,C 180,E1 -14363.176,E2 -14363.176} C_VEL
LIN {X 0,Y 333.611,Z 245.43,A -85,B 0,C 180,E1 -14366.801,E2 -14366.801} C_VEL
LIN {X 0,Y 333.672,Z 245.418,A -85,B 0,C 180,E1 -14369.722,E2 -14369.722} C_VEL
LIN {X 0,Y 333.714,Z 245.413,A -85,B 0,C 180,E1 -14372.41,E2 -14372.41} C_VEL
LIN {X 0,Y 333.709,Z 245.417,A -85,B 0,C 180,E1 -14375.1,E2 -14375.1} C_VEL
LIN {X 0,Y 333.652,Z 245.423,A -85,B 0,C 180,E1 -14379.027,E2 -14379.027} C_VEL
LIN {X 0,Y 333.73,Z 245.415,A -85,B 0,C 180,E1 -14381.596,E2 -14381.596} C_VEL
LIN {X 0,Y 333.803,Z 245.407,A -85,B 0,C 180,E1 -14385.586,E2 -14385.586} C_VEL
LIN {X 0,Y 333.83,Z 245.399,A -85,B 0,C 180,E1 -14389.087,E2 -14389.087} C_VEL
LIN {X 0,Y 333.958,Z 245.381,A -85,B 0,C 180,E1 -14392.755,E2 -14392.755} C_VEL
LIN {X 0,Y 333.792,Z 245.403,A -85,B 0,C 180,E1 -14395.177,E2 -14395.177} C_VEL
LIN {X 0,Y 334.077,Z 245.37,A -85,B 0,C 180,E1 -14397.597,E2 -14397.597} C_VEL
LIN {X 0,Y 334.083,Z 245.366,A -85,B 0,C 180,E1 -14401.213,E2 -14401.213} C_VEL
LIN {X 0,Y 334.073,Z 245.37,A -85,B 0,C 180,E1 -14402.419,E2 -14402.419} C_VEL
LIN {X 0,Y 333.999,Z 245.378,A -85,B 0,C 180,E1 -14406.047,E2 -14406.047} C_VEL
LIN {X 0,Y 333.926,Z 245.391,A -85,B 0,C 180,E1 -14408.479,E2 -14408.479} C_VEL
LIN {X 0,Y 333.805,Z 245.404,A -85,B 0,C 180,E1 -14412.161,E2 -14412.161} C_VEL
LIN {X 0,Y 333.826,Z 245.404,A -85,B 0,C 180,E1 -14414.641,E2 -14414.641} C_VEL
LIN {X 0,Y 333.741,Z 245.414,A -85,B 0,C 180,E1 -14418.622,E2 -14418.622} C_VEL
LIN {X 0,Y 333.673,Z 245.419,A -85,B 0,C 180,E1 -14422.286,E2 -14422.286} C_VEL
LIN {X 0,Y 333.709,Z 245.417,A -85,B 0,C 180,E1 -14425.094,E2 -14425.094} C_VEL
LIN {X 0,Y 333.672,Z 245.423,A -85,B 0,C 180,E1 -14428.983,E2 -14428.983} C_VEL
LIN {X 0,Y 333.667,Z 245.419,A -85,B 0,C 180,E1 -14432.591,E2 -14432.591} C_VEL
LIN {X 0,Y 333.699,Z 245.413,A -85,B 0,C 180,E1 -14436.143,E2 -14436.143} C_VEL
LIN {X 0,Y 333.644,Z 245.425,A -85,B 0,C 180,E1 -14439.2,E2 -14439.2} C_VEL
LIN {X 0,Y 333.63,Z 245.422,A -85,B 0,C 180,E1 -14442.497,E2 -14442.497} C_VEL
LIN {X 0,Y 333.609,Z 245.428,A -85,B 0,C 180,E1 -14445.955,E2 -14445.955} C_VEL
LIN {X 0,Y 333.623,Z 245.426,A -85,B 0,C 180,E1 -14449.328,E2 -14449.328} C_VEL
LIN {X 0,Y 333.686,Z 245.417,A -85,B 0,C 180,E1 -14453.171,E2 -14453.171} C_VEL
LIN {X 0,Y 333.698,Z 245.416,A -85,B 0,C 180,E1 -14455.342,E2 -14455.342} C_VEL
LIN {X 0,Y 333.654,Z 245.426,A -85,B 0,C 180,E1 -14458.222,E2 -14458.222} C_VEL
LIN {X 0,Y 333.696,Z 245.455,A -85,B 0,C 180,E1 -14460.181,E2 -14460.181} C_VEL
LIN {X 0,Y 334.926,Z 251.429,A -85,B 0,C 180,E1 -14462.047,E2 -14462.047} C_VEL
LIN {X 0,Y 336.938,Z 261.694,A -85,B 0,C 180,E1 -14465.013,E2 -14465.013} C_VEL
LIN {X 0,Y 337.33,Z 264.269,A -85,B 0,C 180,E1 -14465.733,E2 -14465.733} C_VEL
LIN {X 0,Y 336.92,Z 268.768,A -85,B 0,C 180,E1 -14466.843,E2 -14466.843} C_VEL
LIN {X 0,Y 342.261,Z 303.162,A -85,B 0,C 180,E1 -14468.033,E2 -14468.033} C_VEL
LIN {X 0,Y 340.52,Z 376.883,A -85,B 0,C 180,E1 -14469.734,E2 -14469.734} C_VEL
LIN {X 0,Y 339.834,Z 390.382,A -85,B 0,C 180,E1 -14470.282,E2 -14470.282} C_VEL
LIN {X 0,Y 339.006,Z 402.743,A -85,B 0,C 180,E1 -14471.019,E2 -14471.019} C_VEL
LIN {X 0,Y 337.935,Z 414.645,A -85,B 0,C 180,E1 -14471.978,E2 -14471.978} C_VEL
LIN {X 0,Y 336.806,Z 426.125,A -85,B 0,C 180,E1 -14473.169,E2 -14473.169} C_VEL
LIN {X 0,Y 335.893,Z 435.977,A -85,B 0,C 180,E1 -14474.449,E2 -14474.449} C_VEL
LIN {X 0,Y 334.756,Z 445.795,A -85,B 0,C 180,E1 -14476.027,E2 -14476.027} C_VEL
LIN {X 0,Y 333.718,Z 454.839,A -85,B 0,C 180,E1 -14477.841,E2 -14477.841} C_VEL
LIN {X 0,Y 333.01,Z 462.099,A -85,B 0,C 180,E1 -14479.664,E2 -14479.664} C_VEL
LIN {X 0,Y 332.504,Z 467.862,A -85,B 0,C 180,E1 -14481.49,E2 -14481.49} C_VEL
LIN {X 0,Y 332.183,Z 472.382,A -85,B 0,C 180,E1 -14483.316,E2 -14483.316} C_VEL
LIN {X 0,Y 331.986,Z 475.787,A -85,B 0,C 180,E1 -14485.14,E2 -14485.14} C_VEL
LIN {X 0,Y 331.966,Z 477.473,A -85,B 0,C 180,E1 -14486.357,E2 -14486.357} C_VEL
LIN {X 0,Y 331.896,Z 478.744,A -85,B 0,C 180,E1 -14487.571,E2 -14487.571} C_VEL
LIN {X 0,Y 331.877,Z 479.6,A -85,B 0,C 180,E1 -14488.785,E2 -14488.785} C_VEL
LIN {X 0,Y 331.896,Z 480.007,A -85,B 0,C 180,E1 -14489.998,E2 -14489.998} C_VEL
LIN {X 0,Y 331.875,Z 480.015,A -85,B 0,C 180,E1 -14491.211,E2 -14491.211} C_VEL
LIN {X 0,Y 331.895,Z 479.63,A -85,B 0,C 180,E1 -14492.425,E2 -14492.425} C_VEL
LIN {X 0,Y 331.969,Z 478.838,A -85,B 0,C 180,E1 -14493.639,E2 -14493.639} C_VEL
LIN {X 0,Y 332.086,Z 476.235,A -85,B 0,C 180,E1 -14495.88,E2 -14495.88} C_VEL
LIN {X 0,Y 332.445,Z 472.646,A -85,B 0,C 180,E1 -14497.896,E2 -14497.896} C_VEL
LIN {X 0,Y 332.977,Z 468.27,A -85,B 0,C 180,E1 -14499.719,E2 -14499.719} C_VEL
LIN {X 0,Y 333.768,Z 462.701,A -85,B 0,C 180,E1 -14501.537,E2 -14501.537} C_VEL
LIN {X 0,Y 334.759,Z 455.759,A -85,B 0,C 180,E1 -14503.35,E2 -14503.35} C_VEL
LIN {X 0,Y 336.192,Z 447.083,A -85,B 0,C 180,E1 -14505.145,E2 -14505.145} C_VEL
LIN {X 0,Y 337.457,Z 437.627,A -85,B 0,C 180,E1 -14506.731,E2 -14506.731} C_VEL
LIN {X 0,Y 338.839,Z 427.329,A -85,B 0,C 180,E1 -14508.124,E2 -14508.124} C_VEL
LIN {X 0,Y 340.311,Z 416.375,A -85,B 0,C 180,E1 -14509.292,E2 -14509.292} C_VEL
LIN {X 0,Y 341.636,Z 404.23,A -85,B 0,C 180,E1 -14510.31,E2 -14510.31} C_VEL
LIN {X 0,Y 342.781,Z 391.604,A -85,B 0,C 180,E1 -14511.103,E2 -14511.103} C_VEL
LIN {X 0,Y 343.703,Z 378.193,A -85,B 0,C 180,E1 -14511.671,E2 -14511.671} C_VEL
LIN {X 0,Y 344.485,Z 357.035,A -85,B 0,C 180,E1 -14512.202,E2 -14512.202} C_VEL
LIN {X 0,Y 345.87,Z 303.46,A -85,B 0,C 180,E1 -14513.467,E2 -14513.467} C_VEL
LIN {X 0,Y 342.758,Z 285.048,A -85,B 0,C 180,E1 -14514.23,E2 -14514.23} C_VEL
LIN {X 0,Y 339.134,Z 269.532,A -85,B 0,C 180,E1 -14514.991,E2 -14514.991} C_VEL
LIN {X 0,Y 338.471,Z 267.359,A -85,B 0,C 180,E1 -14515.168,E2 -14515.168} C_VEL
LIN {X 0,Y 336.668,Z 257.767,A -85,B 0,C 180,E1 -14517.968,E2 -14517.968} C_VEL
LIN {X 0,Y 334.033,Z 246.872,A -85,B 0,C 180,E1 -14521.392,E2 -14521.392} C_VEL
LIN {X 0,Y 333.677,Z 245.45,A -85,B 0,C 180,E1 -14521.98,E2 -14521.98} C_VEL
LIN {X 0,Y 333.697,Z 245.419,A -85,B 0,C 180,E1 -14524.769,E2 -14524.769} C_VEL
LIN {X 0,Y 333.654,Z 245.423,A -85,B 0,C 180,E1 -14527.648,E2 -14527.648} C_VEL
LIN {X 0,Y 333.613,Z 245.427,A -85,B 0,C 180,E1 -14530.769,E2 -14530.769} C_VEL
LIN {X 0,Y 333.597,Z 245.433,A -85,B 0,C 180,E1 -14534.244,E2 -14534.244} C_VEL
LIN {X 0,Y 333.642,Z 245.423,A -85,B 0,C 180,E1 -14537.611,E2 -14537.611} C_VEL
LIN {X 0,Y 333.621,Z 245.425,A -85,B 0,C 180,E1 -14541.205,E2 -14541.205} C_VEL
LIN {X 0,Y 333.677,Z 245.415,A -85,B 0,C 180,E1 -14543.854,E2 -14543.854} C_VEL
LIN {X 0,Y 333.645,Z 245.421,A -85,B 0,C 180,E1 -14547.408,E2 -14547.408} C_VEL
LIN {X 0,Y 333.651,Z 245.422,A -85,B 0,C 180,E1 -14551.015,E2 -14551.015} C_VEL
LIN {X 0,Y 333.697,Z 245.419,A -85,B 0,C 180,E1 -14555.081,E2 -14555.081} C_VEL
LIN {X 0,Y 333.646,Z 245.426,A -85,B 0,C 180,E1 -14559.01,E2 -14559.01} C_VEL
LIN {X 0,Y 333.701,Z 245.415,A -85,B 0,C 180,E1 -14561.577,E2 -14561.577} C_VEL
LIN {X 0,Y 333.767,Z 245.409,A -85,B 0,C 180,E1 -14565.593,E2 -14565.593} C_VEL
LIN {X 0,Y 333.806,Z 245.404,A -85,B 0,C 180,E1 -14569.07,E2 -14569.07} C_VEL
LIN {X 0,Y 333.954,Z 245.387,A -85,B 0,C 180,E1 -14572.738,E2 -14572.738} C_VEL
LIN {X 0,Y 333.773,Z 245.406,A -85,B 0,C 180,E1 -14575.161,E2 -14575.161} C_VEL
LIN {X 0,Y 334.053,Z 245.371,A -85,B 0,C 180,E1 -14577.581,E2 -14577.581} C_VEL
LIN {X 0,Y 334.19,Z 245.352,A -85,B 0,C 180,E1 -14579.992,E2 -14579.992} C_VEL
LIN {X 0,Y 334.086,Z 245.366,A -85,B 0,C 180,E1 -14582.403,E2 -14582.403} C_VEL
LIN {X 0,Y 333.966,Z 245.383,A -85,B 0,C 180,E1 -14586.481,E2 -14586.481} C_VEL
LIN {X 0,Y 333.839,Z 245.404,A -85,B 0,C 180,E1 -14589.687,E2 -14589.687} C_VEL
LIN {X 0,Y 333.767,Z 245.41,A -85,B 0,C 180,E1 -14593.384,E2 -14593.384} C_VEL
LIN {X 0,Y 333.753,Z 245.571,A -85,B 0,C 180,E1 -14596.506,E2 -14596.506} C_VEL
LIN {X 0,Y 335.696,Z 253.181,A -85,B 0,C 180,E1 -14598.926,E2 -14598.926} C_VEL
LIN {X 0,Y 337.156,Z 259.693,A -85,B 0,C 180,E1 -14600.782,E2 -14600.782} C_VEL
LIN {X 0,Y 342.387,Z 272.238,A -85,B 0,C 180,E1 -14601.652,E2 -14601.652} C_VEL
LIN {X 0,Y 346.131,Z 291.025,A -85,B 0,C 180,E1 -14602.486,E2 -14602.486} C_VEL
LIN {X 0,Y 343.892,Z 368.515,A -85,B 0,C 180,E1 -14604.336,E2 -14604.336} C_VEL
LIN {X 0,Y 343.052,Z 382.201,A -85,B 0,C 180,E1 -14604.904,E2 -14604.904} C_VEL
LIN {X 0,Y 342.118,Z 394.093,A -85,B 0,C 180,E1 -14605.627,E2 -14605.627} C_VEL
LIN {X 0,Y 340.828,Z 406.427,A -85,B 0,C 180,E1 -14606.636,E2 -14606.636} C_VEL
LIN {X 0,Y 339.407,Z 417.812,A -85,B 0,C 180,E1 -14607.832,E2 -14607.832} C_VEL
LIN {X 0,Y 337.919,Z 428.568,A -85,B 0,C 180,E1 -14609.264,E2 -14609.264} C_VEL
LIN {X 0,Y 336.6,Z 437.485,A -85,B 0,C 180,E1 -14610.74,E2 -14610.74} C_VEL
LIN {X 0,Y 335.186,Z 446.472,A -85,B 0,C 180,E1 -14612.579,E2 -14612.579} C_VEL
LIN {X 0,Y 334.202,Z 452.886,A -85,B 0,C 180,E1 -14614.219,E2 -14614.219} C_VEL
LIN {X 0,Y 333.297,Z 458.972,A -85,B 0,C 180,E1 -14616.174,E2 -14616.174} C_VEL
LIN {X 0,Y 332.766,Z 462.888,A -85,B 0,C 180,E1 -14617.756,E2 -14617.756} C_VEL
LIN {X 0,Y 332.331,Z 465.986,A -85,B 0,C 180,E1 -14619.364,E2 -14619.364} C_VEL
LIN {X 0,Y 332,Z 468.334,A -85,B 0,C 180,E1 -14620.999,E2 -14620.999} C_VEL
LIN {X 0,Y 331.835,Z 469.943,A -85,B 0,C 180,E1 -14622.652,E2 -14622.652} C_VEL
LIN {X 0,Y 331.7,Z 470.808,A -85,B 0,C 180,E1 -14624.348,E2 -14624.348} C_VEL
LIN {X 0,Y 331.65,Z 470.841,A -85,B 0,C 180,E1 -14626.08,E2 -14626.08} C_VEL
LIN {X 0,Y 331.629,Z 470.019,A -85,B 0,C 180,E1 -14627.863,E2 -14627.863} C_VEL
LIN {X 0,Y 331.788,Z 468.276,A -85,B 0,C 180,E1 -14629.673,E2 -14629.673} C_VEL
LIN {X 0,Y 332.065,Z 465.501,A -85,B 0,C 180,E1 -14631.526,E2 -14631.526} C_VEL
LIN {X 0,Y 332.464,Z 460.853,A -85,B 0,C 180,E1 -14633.712,E2 -14633.712} C_VEL
LIN {X 0,Y 333.002,Z 454.999,A -85,B 0,C 180,E1 -14635.741,E2 -14635.741} C_VEL
LIN {X 0,Y 333.618,Z 448.965,A -85,B 0,C 180,E1 -14637.399,E2 -14637.399} C_VEL
LIN {X 0,Y 334.499,Z 440.852,A -85,B 0,C 180,E1 -14639.197,E2 -14639.197} C_VEL
LIN {X 0,Y 335.553,Z 431.533,A -85,B 0,C 180,E1 -14640.862,E2 -14640.862} C_VEL
LIN {X 0,Y 336.638,Z 421.287,A -85,B 0,C 180,E1 -14642.324,E2 -14642.324} C_VEL
LIN {X 0,Y 337.782,Z 409.853,A -85,B 0,C 180,E1 -14643.627,E2 -14643.627} C_VEL
LIN {X 0,Y 338.756,Z 398.199,A -85,B 0,C 180,E1 -14644.669,E2 -14644.669} C_VEL
LIN {X 0,Y 339.664,Z 385.272,A -85,B 0,C 180,E1 -14645.534,E2 -14645.534} C_VEL
LIN {X 0,Y 340.397,Z 371.92,A -85,B 0,C 180,E1 -14646.16,E2 -14646.16} C_VEL
LIN {X 0,Y 340.92,Z 355.692,A -85,B 0,C 180,E1 -14646.602,E2 -14646.602} C_VEL
LIN {X 0,Y 342.307,Z 289.286,A -85,B 0,C 180,E1 -14648.116,E2 -14648.116} C_VEL
LIN {X 0,Y 337.517,Z 263.473,A -85,B 0,C 180,E1 -14649.02,E2 -14649.02} C_VEL
LIN {X 0,Y 336.458,Z 259.818,A -85,B 0,C 180,E1 -14649.243,E2 -14649.243} C_VEL
LIN {X 0,Y 334.6,Z 249.834,A -85,B 0,C 180,E1 -14652.271,E2 -14652.271} C_VEL
LIN {X 0,Y 333.712,Z 245.462,A -85,B 0,C 180,E1 -14653.721,E2 -14653.721} C_VEL
LIN {X 0,Y 333.724,Z 245.417,A -85,B 0,C 180,E1 -14656.608,E2 -14656.608} C_VEL
LIN {X 0,Y 333.792,Z 245.405,A -85,B 0,C 180,E1 -14660.305,E2 -14660.305} C_VEL
LIN {X 0,Y 333.944,Z 245.39,A -85,B 0,C 180,E1 -14662.748,E2 -14662.748} C_VEL
LIN {X 0,Y 333.752,Z 245.41,A -85,B 0,C 180,E1 -14665.17,E2 -14665.17} C_VEL
LIN {X 0,Y 334.07,Z 245.369,A -85,B 0,C 180,E1 -14667.591,E2 -14667.591} C_VEL
LIN {X 0,Y 334.178,Z 245.354,A -85,B 0,C 180,E1 -14670.002,E2 -14670.002} C_VEL
LIN {X 0,Y 334.071,Z 245.369,A -85,B 0,C 180,E1 -14672.413,E2 -14672.413} C_VEL
LIN {X 0,Y 333.947,Z 245.39,A -85,B 0,C 180,E1 -14677.256,E2 -14677.256} C_VEL
LIN {X 0,Y 333.771,Z 245.406,A -85,B 0,C 180,E1 -14680.926,E2 -14680.926} C_VEL
LIN {X 0,Y 333.745,Z 245.409,A -85,B 0,C 180,E1 -14684.639,E2 -14684.639} C_VEL
LIN {X 0,Y 333.733,Z 245.409,A -85,B 0,C 180,E1 -14688.659,E2 -14688.659} C_VEL
LIN {X 0,Y 333.601,Z 245.428,A -85,B 0,C 180,E1 -14692.286,E2 -14692.286} C_VEL
LIN {X 0,Y 333.679,Z 245.419,A -85,B 0,C 180,E1 -14696.253,E2 -14696.253} C_VEL
LIN {X 0,Y 333.645,Z 245.419,A -85,B 0,C 180,E1 -14698.563,E2 -14698.563} C_VEL
LIN {X 0,Y 332.98,Z 245.505,A -85,B 0,C 180,E1 -14699.57,E2 -14699.57} C_VEL
LIN {X 0,Y 330.095,Z 245.862,A -85,B 0,C 180,E1 -14701.206,E2 -14701.206} C_VEL
LIN {X 0,Y 327.656,Z 246.169,A -85,B 0,C 180,E1 -14702.532,E2 -14702.532} C_VEL
LIN {X 0,Y 326.628,Z 246.296,A -85,B 0,C 180,E1 -14703.559,E2 -14703.559} C_VEL
LIN {X 0,Y 326.555,Z 246.308,A -85,B 0,C 180,E1 -14703.906,E2 -14703.906} C_VEL
LIN {X 0,Y 326.581,Z 246.301,A -85,B 0,C 180,E1 -14707.246,E2 -14707.246} C_VEL
LIN {X 0,Y 326.591,Z 246.303,A -85,B 0,C 180,E1 -14710.211,E2 -14710.211} C_VEL
LIN {X 0,Y 326.617,Z 246.296,A -85,B 0,C 180,E1 -14713.518,E2 -14713.518} C_VEL
LIN {X 0,Y 326.613,Z 246.298,A -85,B 0,C 180,E1 -14717.023,E2 -14717.023} C_VEL
LIN {X 0,Y 326.614,Z 246.303,A -85,B 0,C 180,E1 -14720.775,E2 -14720.775} C_VEL
LIN {X 0,Y 326.585,Z 246.302,A -85,B 0,C 180,E1 -14724.49,E2 -14724.49} C_VEL
LIN {X 0,Y 326.582,Z 246.302,A -85,B 0,C 180,E1 -14727.465,E2 -14727.465} C_VEL
LIN {X 0,Y 326.626,Z 246.296,A -85,B 0,C 180,E1 -14730.349,E2 -14730.349} C_VEL
LIN {X 0,Y 326.672,Z 246.289,A -85,B 0,C 180,E1 -14734.526,E2 -14734.526} C_VEL
LIN {X 0,Y 326.602,Z 246.298,A -85,B 0,C 180,E1 -14738.553,E2 -14738.553} C_VEL
LIN {X 0,Y 326.654,Z 246.291,A -85,B 0,C 180,E1 -14742.479,E2 -14742.479} C_VEL
LIN {X 0,Y 326.754,Z 246.279,A -85,B 0,C 180,E1 -14746.324,E2 -14746.324} C_VEL
LIN {X 0,Y 326.802,Z 246.275,A -85,B 0,C 180,E1 -14750.102,E2 -14750.102} C_VEL
LIN {X 0,Y 326.946,Z 246.26,A -85,B 0,C 180,E1 -14753.839,E2 -14753.839} C_VEL
LIN {X 0,Y 327.021,Z 246.248,A -85,B 0,C 180,E1 -14757.545,E2 -14757.545} C_VEL
LIN {X 0,Y 327.051,Z 246.241,A -85,B 0,C 180,E1 -14761.239,E2 -14761.239} C_VEL
LIN {X 0,Y 326.759,Z 246.278,A -85,B 0,C 180,E1 -14763.707,E2 -14763.707} C_VEL
LIN {X 0,Y 326.953,Z 246.255,A -85,B 0,C 180,E1 -14766.178,E2 -14766.178} C_VEL
LIN {X 0,Y 326.796,Z 246.275,A -85,B 0,C 180,E1 -14769.914,E2 -14769.914} C_VEL
LIN {X 0,Y 326.776,Z 246.277,A -85,B 0,C 180,E1 -14773.692,E2 -14773.692} C_VEL
LIN {X 0,Y 326.682,Z 246.286,A -85,B 0,C 180,E1 -14777.536,E2 -14777.536} C_VEL
LIN {X 0,Y 326.632,Z 246.295,A -85,B 0,C 180,E1 -14781.463,E2 -14781.463} C_VEL
LIN {X 0,Y 326.655,Z 246.293,A -85,B 0,C 180,E1 -14785.494,E2 -14785.494} C_VEL
LIN {X 0,Y 326.611,Z 246.297,A -85,B 0,C 180,E1 -14789.671,E2 -14789.671} C_VEL
LIN {X 0,Y 326.641,Z 246.297,A -85,B 0,C 180,E1 -14792.95,E2 -14792.95} C_VEL
LIN {X 0,Y 326.636,Z 246.296,A -85,B 0,C 180,E1 -14795.524,E2 -14795.524} C_VEL
LIN {X 0,Y 326.611,Z 246.302,A -85,B 0,C 180,E1 -14799.225,E2 -14799.225} C_VEL
LIN {X 0,Y 326.557,Z 246.304,A -85,B 0,C 180,E1 -14802.966,E2 -14802.966} C_VEL
LIN {X 0,Y 326.559,Z 246.304,A -85,B 0,C 180,E1 -14807.039,E2 -14807.039} C_VEL
LIN {X 0,Y 326.597,Z 246.299,A -85,B 0,C 180,E1 -14810.784,E2 -14810.784} C_VEL
LIN {X 0,Y 326.636,Z 246.296,A -85,B 0,C 180,E1 -14814.481,E2 -14814.481} C_VEL
LIN {X 0,Y 326.632,Z 246.297,A -85,B 0,C 180,E1 -14817.456,E2 -14817.456} C_VEL
LIN {X 0,Y 326.706,Z 246.486,A -85,B 0,C 180,E1 -14819.963,E2 -14819.963} C_VEL
LIN {X 0,Y 329.232,Z 258.858,A -85,B 0,C 180,E1 -14823.719,E2 -14823.719} C_VEL
LIN {X 0,Y 330.285,Z 264.952,A -85,B 0,C 180,E1 -14825.483,E2 -14825.483} C_VEL
LIN {X 0,Y 330.066,Z 268.463,A -85,B 0,C 180,E1 -14826.396,E2 -14826.396} C_VEL
LIN {X 0,Y 331.074,Z 275.288,A -85,B 0,C 180,E1 -14826.684,E2 -14826.684} C_VEL
LIN {X 0,Y 335.515,Z 303.577,A -85,B 0,C 180,E1 -14827.654,E2 -14827.654} C_VEL
LIN {X 0,Y 333.804,Z 375.697,A -85,B 0,C 180,E1 -14829.348,E2 -14829.348} C_VEL
LIN {X 0,Y 333.149,Z 388.802,A -85,B 0,C 180,E1 -14829.87,E2 -14829.87} C_VEL
LIN {X 0,Y 332.266,Z 401.534,A -85,B 0,C 180,E1 -14830.619,E2 -14830.619} C_VEL
LIN {X 0,Y 331.177,Z 413.757,A -85,B 0,C 180,E1 -14831.597,E2 -14831.597} C_VEL
LIN {X 0,Y 329.942,Z 425.373,A -85,B 0,C 180,E1 -14832.808,E2 -14832.808} C_VEL
LIN {X 0,Y 328.905,Z 436.25,A -85,B 0,C 180,E1 -14834.244,E2 -14834.244} C_VEL
LIN {X 0,Y 327.801,Z 445.288,A -85,B 0,C 180,E1 -14835.724,E2 -14835.724} C_VEL
LIN {X 0,Y 326.942,Z 453.03,A -85,B 0,C 180,E1 -14837.269,E2 -14837.269} C_VEL
LIN {X 0,Y 326.106,Z 460.604,A -85,B 0,C 180,E1 -14839.128,E2 -14839.128} C_VEL
LIN {X 0,Y 325.443,Z 467.568,A -85,B 0,C 180,E1 -14841.303,E2 -14841.303} C_VEL
LIN {X 0,Y 325.105,Z 472.135,A -85,B 0,C 180,E1 -14843.17,E2 -14843.17} C_VEL
LIN {X 0,Y 324.902,Z 475.584,A -85,B 0,C 180,E1 -14845.034,E2 -14845.034} C_VEL
LIN {X 0,Y 324.874,Z 477.29,A -85,B 0,C 180,E1 -14846.277,E2 -14846.277} C_VEL
LIN {X 0,Y 324.817,Z 478.58,A -85,B 0,C 180,E1 -14847.518,E2 -14847.518} C_VEL
LIN {X 0,Y 324.789,Z 479.463,A -85,B 0,C 180,E1 -14848.758,E2 -14848.758} C_VEL
LIN {X 0,Y 324.805,Z 479.898,A -85,B 0,C 180,E1 -14849.998,E2 -14849.998} C_VEL
LIN {X 0,Y 324.787,Z 479.925,A -85,B 0,C 180,E1 -14851.238,E2 -14851.238} C_VEL
LIN {X 0,Y 324.817,Z 479.559,A -85,B 0,C 180,E1 -14852.478,E2 -14852.478} C_VEL
LIN {X 0,Y 324.879,Z 478.798,A -85,B 0,C 180,E1 -14853.719,E2 -14853.719} C_VEL
LIN {X 0,Y 325.006,Z 476.478,A -85,B 0,C 180,E1 -14855.853,E2 -14855.853} C_VEL
LIN {X 0,Y 325.409,Z 472.702,A -85,B 0,C 180,E1 -14858.068,E2 -14858.068} C_VEL
LIN {X 0,Y 325.962,Z 468.368,A -85,B 0,C 180,E1 -14859.93,E2 -14859.93} C_VEL
LIN {X 0,Y 326.913,Z 461.821,A -85,B 0,C 180,E1 -14862.097,E2 -14862.097} C_VEL
LIN {X 0,Y 328.113,Z 454.647,A -85,B 0,C 180,E1 -14863.941,E2 -14863.941} C_VEL
LIN {X 0,Y 329.591,Z 445.726,A -85,B 0,C 180,E1 -14865.773,E2 -14865.773} C_VEL
LIN {X 0,Y 330.878,Z 436.642,A -85,B 0,C 180,E1 -14867.297,E2 -14867.297} C_VEL
LIN {X 0,Y 332.347,Z 426.631,A -85,B 0,C 180,E1 -14868.651,E2 -14868.651} C_VEL
LIN {X 0,Y 333.885,Z 415.559,A -85,B 0,C 180,E1 -14869.839,E2 -14869.839} C_VEL
LIN {X 0,Y 335.036,Z 405.21,A -85,B 0,C 180,E1 -14870.729,E2 -14870.729} C_VEL
LIN {X 0,Y 336.245,Z 392.938,A -85,B 0,C 180,E1 -14871.533,E2 -14871.533} C_VEL
LIN {X 0,Y 337.184,Z 380.443,A -85,B 0,C 180,E1 -14872.113,E2 -14872.113} C_VEL
LIN {X 0,Y 337.905,Z 364.836,A -85,B 0,C 180,E1 -14872.547,E2 -14872.547} C_VEL
LIN {X 0,Y 339.589,Z 304.487,A -85,B 0,C 180,E1 -14873.997,E2 -14873.997} C_VEL
LIN {X 0,Y 336.334,Z 285.435,A -85,B 0,C 180,E1 -14874.823,E2 -14874.823} C_VEL
LIN {X 0,Y 333.208,Z 272.023,A -85,B 0,C 180,E1 -14875.514,E2 -14875.514} C_VEL
LIN {X 0,Y 331.363,Z 267.293,A -85,B 0,C 180,E1 -14875.878,E2 -14875.878} C_VEL
LIN {X 0,Y 329.517,Z 258.054,A -85,B 0,C 180,E1 -14878.666,E2 -14878.666} C_VEL
LIN {X 0,Y 327.205,Z 248.589,A -85,B 0,C 180,E1 -14881.748,E2 -14881.748} C_VEL
LIN {X 0,Y 326.626,Z 246.349,A -85,B 0,C 180,E1 -14882.61,E2 -14882.61} C_VEL
LIN {X 0,Y 326.624,Z 246.301,A -85,B 0,C 180,E1 -14885.515,E2 -14885.515} C_VEL
LIN {X 0,Y 326.582,Z 246.303,A -85,B 0,C 180,E1 -14889.213,E2 -14889.213} C_VEL
LIN {X 0,Y 326.58,Z 246.302,A -85,B 0,C 180,E1 -14892.965,E2 -14892.965} C_VEL
LIN {X 0,Y 326.579,Z 246.304,A -85,B 0,C 180,E1 -14897.024,E2 -14897.024} C_VEL
LIN {X 0,Y 326.577,Z 246.301,A -85,B 0,C 180,E1 -14900.776,E2 -14900.776} C_VEL
LIN {X 0,Y 326.614,Z 246.298,A -85,B 0,C 180,E1 -14904.474,E2 -14904.474} C_VEL
LIN {X 0,Y 326.609,Z 246.297,A -85,B 0,C 180,E1 -14907.449,E2 -14907.449} C_VEL
LIN {X 0,Y 326.591,Z 246.297,A -85,B 0,C 180,E1 -14910.327,E2 -14910.327} C_VEL
LIN {X 0,Y 326.634,Z 246.293,A -85,B 0,C 180,E1 -14914.505,E2 -14914.505} C_VEL
LIN {X 0,Y 326.605,Z 246.3,A -85,B 0,C 180,E1 -14918.535,E2 -14918.535} C_VEL
LIN {X 0,Y 326.618,Z 246.3,A -85,B 0,C 180,E1 -14922.46,E2 -14922.46} C_VEL
LIN {X 0,Y 326.737,Z 246.285,A -85,B 0,C 180,E1 -14926.306,E2 -14926.306} C_VEL
LIN {X 0,Y 326.772,Z 246.28,A -85,B 0,C 180,E1 -14930.085,E2 -14930.085} C_VEL
LIN {X 0,Y 326.938,Z 246.255,A -85,B 0,C 180,E1 -14933.822,E2 -14933.822} C_VEL
LIN {X 0,Y 326.996,Z 246.249,A -85,B 0,C 180,E1 -14937.528,E2 -14937.528} C_VEL
LIN {X 0,Y 327.143,Z 246.23,A -85,B 0,C 180,E1 -14939.992,E2 -14939.992} C_VEL
LIN {X 0,Y 327.026,Z 246.245,A -85,B 0,C 180,E1 -14942.455,E2 -14942.455} C_VEL
LIN {X 0,Y 326.94,Z 246.259,A -85,B 0,C 180,E1 -14946.47,E2 -14946.47} C_VEL
LIN {X 0,Y 326.892,Z 246.266,A -85,B 0,C 180,E1 -14948.647,E2 -14948.647} C_VEL
LIN {X 0,Y 326.711,Z 246.288,A -85,B 0,C 180,E1 -14952.413,E2 -14952.413} C_VEL
LIN {X 0,Y 326.737,Z 246.415,A -85,B 0,C 180,E1 -14955.828,E2 -14955.828} C_VEL
LIN {X 0,Y 329.187,Z 256.122,A -85,B 0,C 180,E1 -14958.991,E2 -14958.991} C_VEL
LIN {X 0,Y 330,Z 259.726,A -85,B 0,C 180,E1 -14960.037,E2 -14960.037} C_VEL
LIN {X 0,Y 336.445,Z 274.734,A -85,B 0,C 180,E1 -14961.149,E2 -14961.149} C_VEL
LIN {X 0,Y 339.887,Z 292.319,A -85,B 0,C 180,E1 -14961.961,E2 -14961.961} C_VEL
LIN {X 0,Y 337.537,Z 368.222,A -85,B 0,C 180,E1 -14963.801,E2 -14963.801} C_VEL
LIN {X 0,Y 336.639,Z 381.997,A -85,B 0,C 180,E1 -14964.375,E2 -14964.375} C_VEL
LIN {X 0,Y 335.625,Z 394.607,A -85,B 0,C 180,E1 -14965.158,E2 -14965.158} C_VEL
LIN {X 0,Y 334.265,Z 406.917,A -85,B 0,C 180,E1 -14966.191,E2 -14966.191} C_VEL
LIN {X 0,Y 332.685,Z 418.798,A -85,B 0,C 180,E1 -14967.476,E2 -14967.476} C_VEL
LIN {X 0,Y 331.22,Z 428.79,A -85,B 0,C 180,E1 -14968.852,E2 -14968.852} C_VEL
LIN {X 0,Y 329.775,Z 437.93,A -85,B 0,C 180,E1 -14970.405,E2 -14970.405} C_VEL
LIN {X 0,Y 328.474,Z 445.894,A -85,B 0,C 180,E1 -14972.065,E2 -14972.065} C_VEL
LIN {X 0,Y 327.28,Z 453.119,A -85,B 0,C 180,E1 -14973.927,E2 -14973.927} C_VEL
LIN {X 0,Y 326.324,Z 459.139,A -85,B 0,C 180,E1 -14975.909,E2 -14975.909} C_VEL
LIN {X 0,Y 325.615,Z 463.9,A -85,B 0,C 180,E1 -14977.948,E2 -14977.948} C_VEL
LIN {X 0,Y 325.17,Z 466.887,A -85,B 0,C 180,E1 -14979.647,E2 -14979.647} C_VEL
LIN {X 0,Y 324.784,Z 469.751,A -85,B 0,C 180,E1 -14982.115,E2 -14982.115} C_VEL
LIN {X 0,Y 324.596,Z 470.943,A -85,B 0,C 180,E1 -14984.402,E2 -14984.402} C_VEL
LIN {X 0,Y 324.545,Z 470.922,A -85,B 0,C 180,E1 -14986.139,E2 -14986.139} C_VEL
LIN {X 0,Y 324.536,Z 470.114,A -85,B 0,C 180,E1 -14987.835,E2 -14987.835} C_VEL
LIN {X 0,Y 324.683,Z 468.578,A -85,B 0,C 180,E1 -14989.509,E2 -14989.509} C_VEL
LIN {X 0,Y 324.898,Z 466.332,A -85,B 0,C 180,E1 -14991.151,E2 -14991.151} C_VEL
LIN {X 0,Y 325.216,Z 462.667,A -85,B 0,C 180,E1 -14993.071,E2 -14993.071} C_VEL
LIN {X 0,Y 325.712,Z 457.588,A -85,B 0,C 180,E1 -14995.059,E2 -14995.059} C_VEL
LIN {X 0,Y 326.404,Z 450.885,A -85,B 0,C 180,E1 -14997.091,E2 -14997.091} C_VEL
LIN {X 0,Y 327.242,Z 443.038,A -85,B 0,C 180,E1 -14998.976,E2 -14998.976} C_VEL
LIN {X 0,Y 328.337,Z 433.968,A -85,B 0,C 180,E1 -15000.706,E2 -15000.706} C_VEL
LIN {X 0,Y 329.361,Z 424.543,A -85,B 0,C 180,E1 -15002.168,E2 -15002.168} C_VEL
LIN {X 0,Y 330.511,Z 414.085,A -85,B 0,C 180,E1 -15003.481,E2 -15003.481} C_VEL
LIN {X 0,Y 331.528,Z 403.074,A -85,B 0,C 180,E1 -15004.581,E2 -15004.581} C_VEL
LIN {X 0,Y 332.481,Z 390.736,A -85,B 0,C 180,E1 -15005.534,E2 -15005.534} C_VEL
LIN {X 0,Y 333.336,Z 377.657,A -85,B 0,C 180,E1 -15006.27,E2 -15006.27} C_VEL
LIN {X 0,Y 333.886,Z 364.701,A -85,B 0,C 180,E1 -15006.742,E2 -15006.742} C_VEL
LIN {X 0,Y 335.607,Z 290.301,A -85,B 0,C 180,E1 -15008.479,E2 -15008.479} C_VEL
LIN {X 0,Y 331.196,Z 266.09,A -85,B 0,C 180,E1 -15009.345,E2 -15009.345} C_VEL
LIN {X 0,Y 329.284,Z 260.012,A -85,B 0,C 180,E1 -15009.672,E2 -15009.672} C_VEL
LIN {X 0,Y 327.553,Z 250.789,A -85,B 0,C 180,E1 -15012.522,E2 -15012.522} C_VEL
LIN {X 0,Y 326.673,Z 246.331,A -85,B 0,C 180,E1 -15014.042,E2 -15014.042} C_VEL
LIN {X 0,Y 326.667,Z 246.291,A -85,B 0,C 180,E1 -15017.578,E2 -15017.578} C_VEL
LIN {X 0,Y 326.845,Z 246.269,A -85,B 0,C 180,E1 -15021.457,E2 -15021.457} C_VEL
LIN {X 0,Y 326.923,Z 246.259,A -85,B 0,C 180,E1 -15023.832,E2 -15023.832} C_VEL
LIN {X 0,Y 327.008,Z 246.249,A -85,B 0,C 180,E1 -15027.539,E2 -15027.539} C_VEL
LIN {X 0,Y 327.13,Z 246.232,A -85,B 0,C 180,E1 -15030.002,E2 -15030.002} C_VEL
LIN {X 0,Y 327.008,Z 246.249,A -85,B 0,C 180,E1 -15032.466,E2 -15032.466} C_VEL
LIN {X 0,Y 326.925,Z 246.258,A -85,B 0,C 180,E1 -15036.172,E2 -15036.172} C_VEL
LIN {X 0,Y 326.748,Z 246.28,A -85,B 0,C 180,E1 -15039.91,E2 -15039.91} C_VEL
LIN {X 0,Y 326.693,Z 246.291,A -85,B 0,C 180,E1 -15043.69,E2 -15043.69} C_VEL
LIN {X 0,Y 326.636,Z 246.299,A -85,B 0,C 180,E1 -15047.533,E2 -15047.533} C_VEL
LIN {X 0,Y 326.596,Z 246.3,A -85,B 0,C 180,E1 -15050.141,E2 -15050.141} C_VEL
LIN {X 0,Y 326.593,Z 246.302,A -85,B 0,C 180,E1 -15054.135,E2 -15054.135} C_VEL
LIN {X 0,Y 326.629,Z 246.293,A -85,B 0,C 180,E1 -15056.865,E2 -15056.865} C_VEL
LIN {X 0,Y 326.589,Z 246.3,A -85,B 0,C 180,E1 -15060.619,E2 -15060.619} C_VEL
LIN {X 0,Y 326.555,Z 246.308,A -85,B 0,C 180,E1 -15063.906,E2 -15063.906} C_VEL
LIN {X 0,Y 325.905,Z 246.394,A -85,B 0,C 180,E1 -15064.936,E2 -15064.936} C_VEL
LIN {X 0,Y 323.029,Z 246.749,A -85,B 0,C 180,E1 -15066.611,E2 -15066.611} C_VEL
LIN {X 0,Y 320.598,Z 247.049,A -85,B 0,C 180,E1 -15067.968,E2 -15067.968} C_VEL
LIN {X 0,Y 319.587,Z 247.172,A -85,B 0,C 180,E1 -15069.02,E2 -15069.02} C_VEL
LIN {X 0,Y 319.522,Z 247.178,A -85,B 0,C 180,E1 -15069.376,E2 -15069.376} C_VEL
LIN {X 0,Y 319.585,Z 247.174,A -85,B 0,C 180,E1 -15072.981,E2 -15072.981} C_VEL
LIN {X 0,Y 319.593,Z 247.176,A -85,B 0,C 180,E1 -15076.528,E2 -15076.528} C_VEL
LIN {X 0,Y 319.553,Z 247.179,A -85,B 0,C 180,E1 -15080.386,E2 -15080.386} C_VEL
LIN {X 0,Y 319.532,Z 247.178,A -85,B 0,C 180,E1 -15083.582,E2 -15083.582} C_VEL
LIN {X 0,Y 319.552,Z 247.179,A -85,B 0,C 180,E1 -15086.696,E2 -15086.696} C_VEL
LIN {X 0,Y 319.562,Z 247.176,A -85,B 0,C 180,E1 -15089.625,E2 -15089.625} C_VEL
LIN {X 0,Y 319.582,Z 247.173,A -85,B 0,C 180,E1 -15092.507,E2 -15092.507} C_VEL
LIN {X 0,Y 319.587,Z 247.177,A -85,B 0,C 180,E1 -15095.314,E2 -15095.314} C_VEL
LIN {X 0,Y 319.565,Z 247.181,A -85,B 0,C 180,E1 -15099.408,E2 -15099.408} C_VEL
LIN {X 0,Y 319.643,Z 247.169,A -85,B 0,C 180,E1 -15103.401,E2 -15103.401} C_VEL
LIN {X 0,Y 319.727,Z 247.156,A -85,B 0,C 180,E1 -15106.017,E2 -15106.017} C_VEL
LIN {X 0,Y 319.75,Z 247.156,A -85,B 0,C 180,E1 -15109.882,E2 -15109.882} C_VEL
LIN {X 0,Y 319.902,Z 247.136,A -85,B 0,C 180,E1 -15113.702,E2 -15113.702} C_VEL
LIN {X 0,Y 319.967,Z 247.127,A -85,B 0,C 180,E1 -15117.491,E2 -15117.491} C_VEL
LIN {X 0,Y 320.019,Z 247.117,A -85,B 0,C 180,E1 -15121.267,E2 -15121.267} C_VEL
LIN {X 0,Y 319.727,Z 247.148,A -85,B 0,C 180,E1 -15125.052,E2 -15125.052} C_VEL
LIN {X 0,Y 319.865,Z 247.135,A -85,B 0,C 180,E1 -15127.583,E2 -15127.583} C_VEL
LIN {X 0,Y 319.729,Z 247.154,A -85,B 0,C 180,E1 -15131.418,E2 -15131.418} C_VEL
LIN {X 0,Y 319.729,Z 247.158,A -85,B 0,C 180,E1 -15134.717,E2 -15134.717} C_VEL
LIN {X 0,Y 319.632,Z 247.164,A -85,B 0,C 180,E1 -15137.936,E2 -15137.936} C_VEL
LIN {X 0,Y 319.585,Z 247.172,A -85,B 0,C 180,E1 -15141.96,E2 -15141.96} C_VEL
LIN {X 0,Y 319.589,Z 247.172,A -85,B 0,C 180,E1 -15146.099,E2 -15146.099} C_VEL
LIN {X 0,Y 319.553,Z 247.179,A -85,B 0,C 180,E1 -15148.944,E2 -15148.944} C_VEL
LIN {X 0,Y 319.548,Z 247.178,A -85,B 0,C 180,E1 -15151.867,E2 -15151.867} C_VEL
LIN {X 0,Y 319.604,Z 247.171,A -85,B 0,C 180,E1 -15155.546,E2 -15155.546} C_VEL
LIN {X 0,Y 319.554,Z 247.18,A -85,B 0,C 180,E1 -15159.665,E2 -15159.665} C_VEL
LIN {X 0,Y 319.509,Z 247.186,A -85,B 0,C 180,E1 -15163.456,E2 -15163.456} C_VEL
LIN {X 0,Y 319.513,Z 247.181,A -85,B 0,C 180,E1 -15167.007,E2 -15167.007} C_VEL
LIN {X 0,Y 319.542,Z 247.179,A -85,B 0,C 180,E1 -15170.368,E2 -15170.368} C_VEL
LIN {X 0,Y 319.604,Z 247.172,A -85,B 0,C 180,E1 -15174.46,E2 -15174.46} C_VEL
LIN {X 0,Y 319.549,Z 247.182,A -85,B 0,C 180,E1 -15178.138,E2 -15178.138} C_VEL
LIN {X 0,Y 319.629,Z 247.331,A -85,B 0,C 180,E1 -15179.619,E2 -15179.619} C_VEL
LIN {X 0,Y 322.165,Z 259.632,A -85,B 0,C 180,E1 -15183.443,E2 -15183.443} C_VEL
LIN {X 0,Y 323.322,Z 266.945,A -85,B 0,C 180,E1 -15185.605,E2 -15185.605} C_VEL
LIN {X 0,Y 323.221,Z 268.441,A -85,B 0,C 180,E1 -15185.967,E2 -15185.967} C_VEL
LIN {X 0,Y 324.723,Z 278.335,A -85,B 0,C 180,E1 -15186.368,E2 -15186.368} C_VEL
LIN {X 0,Y 328.789,Z 304.632,A -85,B 0,C 180,E1 -15187.291,E2 -15187.291} C_VEL
LIN {X 0,Y 326.979,Z 376.35,A -85,B 0,C 180,E1 -15189.02,E2 -15189.02} C_VEL
LIN {X 0,Y 326.239,Z 389.925,A -85,B 0,C 180,E1 -15189.589,E2 -15189.589} C_VEL
LIN {X 0,Y 325.365,Z 402.351,A -85,B 0,C 180,E1 -15190.355,E2 -15190.355} C_VEL
LIN {X 0,Y 324.241,Z 414.307,A -85,B 0,C 180,E1 -15191.353,E2 -15191.353} C_VEL
LIN {X 0,Y 322.975,Z 425.807,A -85,B 0,C 180,E1 -15192.588,E2 -15192.588} C_VEL
LIN {X 0,Y 321.916,Z 436.528,A -85,B 0,C 180,E1 -15194.048,E2 -15194.048} C_VEL
LIN {X 0,Y 320.684,Z 446.365,A -85,B 0,C 180,E1 -15195.724,E2 -15195.724} C_VEL
LIN {X 0,Y 319.607,Z 455.29,A -85,B 0,C 180,E1 -15197.618,E2 -15197.618} C_VEL
LIN {X 0,Y 318.844,Z 462.395,A -85,B 0,C 180,E1 -15199.521,E2 -15199.521} C_VEL
LIN {X 0,Y 318.244,Z 468.885,A -85,B 0,C 180,E1 -15201.745,E2 -15201.745} C_VEL
LIN {X 0,Y 317.938,Z 473.126,A -85,B 0,C 180,E1 -15203.652,E2 -15203.652} C_VEL
LIN {X 0,Y 317.823,Z 475.357,A -85,B 0,C 180,E1 -15204.923,E2 -15204.923} C_VEL
LIN {X 0,Y 317.786,Z 477.09,A -85,B 0,C 180,E1 -15206.194,E2 -15206.194} C_VEL
LIN {X 0,Y 317.741,Z 478.403,A -85,B 0,C 180,E1 -15207.462,E2 -15207.462} C_VEL
LIN {X 0,Y 317.703,Z 479.311,A -85,B 0,C 180,E1 -15208.73,E2 -15208.73} C_VEL
LIN {X 0,Y 317.716,Z 479.787,A -85,B 0,C 180,E1 -15209.998,E2 -15209.998} C_VEL
LIN {X 0,Y 317.702,Z 479.836,A -85,B 0,C 180,E1 -15211.265,E2 -15211.265} C_VEL
LIN {X 0,Y 317.74,Z 479.491,A -85,B 0,C 180,E1 -15212.533,E2 -15212.533} C_VEL
LIN {X 0,Y 317.791,Z 478.753,A -85,B 0,C 180,E1 -15213.802,E2 -15213.802} C_VEL
LIN {X 0,Y 317.905,Z 476.739,A -85,B 0,C 180,E1 -15215.788,E2 -15215.788} C_VEL
LIN {X 0,Y 318.203,Z 473.948,A -85,B 0,C 180,E1 -15217.613,E2 -15217.613} C_VEL
LIN {X 0,Y 318.725,Z 470.025,A -85,B 0,C 180,E1 -15219.517,E2 -15219.517} C_VEL
LIN {X 0,Y 319.496,Z 464.969,A -85,B 0,C 180,E1 -15221.416,E2 -15221.416} C_VEL
LIN {X 0,Y 320.523,Z 458.644,A -85,B 0,C 180,E1 -15223.308,E2 -15223.308} C_VEL
LIN {X 0,Y 321.987,Z 450.734,A -85,B 0,C 180,E1 -15225.182,E2 -15225.182} C_VEL
LIN {X 0,Y 323.43,Z 441.562,A -85,B 0,C 180,E1 -15226.938,E2 -15226.938} C_VEL
LIN {X 0,Y 324.903,Z 431.864,A -85,B 0,C 180,E1 -15228.44,E2 -15228.44} C_VEL
LIN {X 0,Y 326.586,Z 420.682,A -85,B 0,C 180,E1 -15229.809,E2 -15229.809} C_VEL
LIN {X 0,Y 328.201,Z 408.067,A -85,B 0,C 180,E1 -15231.017,E2 -15231.017} C_VEL
LIN {X 0,Y 329.653,Z 395.486,A -85,B 0,C 180,E1 -15231.904,E2 -15231.904} C_VEL
LIN {X 0,Y 330.663,Z 382.36,A -85,B 0,C 180,E1 -15232.573,E2 -15232.573} C_VEL
LIN {X 0,Y 331.423,Z 369.856,A -85,B 0,C 180,E1 -15232.971,E2 -15232.971} C_VEL
LIN {X 0,Y 333.287,Z 305.146,A -85,B 0,C 180,E1 -15234.571,E2 -15234.571} C_VEL
LIN {X 0,Y 330.331,Z 287.563,A -85,B 0,C 180,E1 -15235.361,E2 -15235.361} C_VEL
LIN {X 0,Y 327.357,Z 274.592,A -85,B 0,C 180,E1 -15236.049,E2 -15236.049} C_VEL
LIN {X 0,Y 324.257,Z 267.198,A -85,B 0,C 180,E1 -15236.641,E2 -15236.641} C_VEL
LIN {X 0,Y 322.423,Z 258.661,A -85,B 0,C 180,E1 -15239.311,E2 -15239.311} C_VEL
LIN {X 0,Y 320.366,Z 250.292,A -85,B 0,C 180,E1 -15242.136,E2 -15242.136} C_VEL
LIN {X 0,Y 319.592,Z 247.238,A -85,B 0,C 180,E1 -15243.308,E2 -15243.308} C_VEL
LIN {X 0,Y 319.568,Z 247.179,A -85,B 0,C 180,E1 -15246.423,E2 -15246.423} C_VEL
LIN {X 0,Y 319.54,Z 247.181,A -85,B 0,C 180,E1 -15249.657,E2 -15249.657} C_VEL
LIN {X 0,Y 319.527,Z 247.18,A -85,B 0,C 180,E1 -15253.454,E2 -15253.454} C_VEL
LIN {X 0,Y 319.557,Z 247.179,A -85,B 0,C 180,E1 -15257.009,E2 -15257.009} C_VEL
LIN {X 0,Y 319.522,Z 247.18,A -85,B 0,C 180,E1 -15260.36,E2 -15260.36} C_VEL
LIN {X 0,Y 319.582,Z 247.173,A -85,B 0,C 180,E1 -15264.452,E2 -15264.452} C_VEL
LIN {X 0,Y 319.526,Z 247.182,A -85,B 0,C 180,E1 -15268.13,E2 -15268.13} C_VEL
LIN {X 0,Y 319.569,Z 247.177,A -85,B 0,C 180,E1 -15271.598,E2 -15271.598} C_VEL
LIN {X 0,Y 319.572,Z 247.178,A -85,B 0,C 180,E1 -15275.294,E2 -15275.294} C_VEL
LIN {X 0,Y 319.56,Z 247.174,A -85,B 0,C 180,E1 -15278.038,E2 -15278.038} C_VEL
LIN {X 0,Y 319.57,Z 247.176,A -85,B 0,C 180,E1 -15282.061,E2 -15282.061} C_VEL
LIN {X 0,Y 319.703,Z 247.161,A -85,B 0,C 180,E1 -15285.999,E2 -15285.999} C_VEL
LIN {X 0,Y 319.725,Z 247.158,A -85,B 0,C 180,E1 -15289.864,E2 -15289.864} C_VEL
LIN {X 0,Y 319.895,Z 247.133,A -85,B 0,C 180,E1 -15293.686,E2 -15293.686} C_VEL
LIN {X 0,Y 320.003,Z 247.125,A -85,B 0,C 180,E1 -15298.733,E2 -15298.733} C_VEL
LIN {X 0,Y 320.001,Z 247.126,A -85,B 0,C 180,E1 -15301.25,E2 -15301.25} C_VEL
LIN {X 0,Y 319.719,Z 247.161,A -85,B 0,C 180,E1 -15303.773,E2 -15303.773} C_VEL
LIN {X 0,Y 319.905,Z 247.136,A -85,B 0,C 180,E1 -15306.457,E2 -15306.457} C_VEL
LIN {X 0,Y 319.819,Z 247.146,A -85,B 0,C 180,E1 -15308.84,E2 -15308.84} C_VEL
LIN {X 0,Y 319.657,Z 247.168,A -85,B 0,C 180,E1 -15312.691,E2 -15312.691} C_VEL
LIN {X 0,Y 319.693,Z 247.249,A -85,B 0,C 180,E1 -15315.073,E2 -15315.073} C_VEL
LIN {X 0,Y 321.219,Z 253.203,A -85,B 0,C 180,E1 -15317.17,E2 -15317.17} C_VEL
LIN {X 0,Y 322.834,Z 259.884,A -85,B 0,C 180,E1 -15319.255,E2 -15319.255} C_VEL
LIN {X 0,Y 329.225,Z 274.081,A -85,B 0,C 180,E1 -15320.395,E2 -15320.395} C_VEL
LIN {X 0,Y 330.735,Z 278.117,A -85,B 0,C 180,E1 -15320.67,E2 -15320.67} C_VEL
LIN {X 0,Y 333.654,Z 293.381,A -85,B 0,C 180,E1 -15321.392,E2 -15321.392} C_VEL
LIN {X 0,Y 331.179,Z 368.66,A -85,B 0,C 180,E1 -15323.271,E2 -15323.271} C_VEL
LIN {X 0,Y 330.284,Z 381.946,A -85,B 0,C 180,E1 -15323.836,E2 -15323.836} C_VEL
LIN {X 0,Y 329.231,Z 394.045,A -85,B 0,C 180,E1 -15324.588,E2 -15324.588} C_VEL
LIN {X 0,Y 327.827,Z 406.325,A -85,B 0,C 180,E1 -15325.619,E2 -15325.619} C_VEL
LIN {X 0,Y 326.247,Z 417.98,A -85,B 0,C 180,E1 -15326.885,E2 -15326.885} C_VEL
LIN {X 0,Y 324.79,Z 427.743,A -85,B 0,C 180,E1 -15328.218,E2 -15328.218} C_VEL
LIN {X 0,Y 323.261,Z 436.873,A -85,B 0,C 180,E1 -15329.757,E2 -15329.757} C_VEL
LIN {X 0,Y 321.737,Z 445.705,A -85,B 0,C 180,E1 -15331.606,E2 -15331.606} C_VEL
LIN {X 0,Y 320.418,Z 453.118,A -85,B 0,C 180,E1 -15333.547,E2 -15333.547} C_VEL
LIN {X 0,Y 319.425,Z 458.995,A -85,B 0,C 180,E1 -15335.509,E2 -15335.509} C_VEL
LIN {X 0,Y 318.675,Z 463.532,A -85,B 0,C 180,E1 -15337.45,E2 -15337.45} C_VEL
LIN {X 0,Y 318.049,Z 467.573,A -85,B 0,C 180,E1 -15339.839,E2 -15339.839} C_VEL
LIN {X 0,Y 317.742,Z 469.51,A -85,B 0,C 180,E1 -15341.557,E2 -15341.557} C_VEL
LIN {X 0,Y 317.583,Z 470.711,A -85,B 0,C 180,E1 -15343.301,E2 -15343.301} C_VEL
LIN {X 0,Y 317.466,Z 471.138,A -85,B 0,C 180,E1 -15345.09,E2 -15345.09} C_VEL
LIN {X 0,Y 317.424,Z 470.711,A -85,B 0,C 180,E1 -15346.924,E2 -15346.924} C_VEL
LIN {X 0,Y 317.499,Z 469.398,A -85,B 0,C 180,E1 -15348.799,E2 -15348.799} C_VEL
LIN {X 0,Y 317.731,Z 467.112,A -85,B 0,C 180,E1 -15350.712,E2 -15350.712} C_VEL
LIN {X 0,Y 318.042,Z 463.692,A -85,B 0,C 180,E1 -15352.685,E2 -15352.685} C_VEL
LIN {X 0,Y 318.512,Z 458.963,A -85,B 0,C 180,E1 -15354.707,E2 -15354.707} C_VEL
LIN {X 0,Y 319.201,Z 452.693,A -85,B 0,C 180,E1 -15356.768,E2 -15356.768} C_VEL
LIN {X 0,Y 320.079,Z 444.398,A -85,B 0,C 180,E1 -15358.884,E2 -15358.884} C_VEL
LIN {X 0,Y 321.234,Z 435.169,A -85,B 0,C 180,E1 -15360.745,E2 -15360.745} C_VEL
LIN {X 0,Y 322.398,Z 424.791,A -85,B 0,C 180,E1 -15362.407,E2 -15362.407} C_VEL
LIN {X 0,Y 323.598,Z 414.425,A -85,B 0,C 180,E1 -15363.739,E2 -15363.739} C_VEL
LIN {X 0,Y 324.724,Z 402.572,A -85,B 0,C 180,E1 -15364.943,E2 -15364.943} C_VEL
LIN {X 0,Y 325.667,Z 390.569,A -85,B 0,C 180,E1 -15365.881,E2 -15365.881} C_VEL
LIN {X 0,Y 326.532,Z 377.575,A -85,B 0,C 180,E1 -15366.622,E2 -15366.622} C_VEL
LIN {X 0,Y 327.141,Z 363.596,A -85,B 0,C 180,E1 -15367.128,E2 -15367.128} C_VEL
LIN {X 0,Y 328.895,Z 291.415,A -85,B 0,C 180,E1 -15368.856,E2 -15368.856} C_VEL
LIN {X 0,Y 324.575,Z 267.545,A -85,B 0,C 180,E1 -15369.732,E2 -15369.732} C_VEL
LIN {X 0,Y 322.156,Z 260.276,A -85,B 0,C 180,E1 -15370.113,E2 -15370.113} C_VEL
LIN {X 0,Y 320.519,Z 251.736,A -85,B 0,C 180,E1 -15372.784,E2 -15372.784} C_VEL
LIN {X 0,Y 319.64,Z 247.228,A -85,B 0,C 180,E1 -15374.336,E2 -15374.336} C_VEL
LIN {X 0,Y 319.613,Z 247.171,A -85,B 0,C 180,E1 -15377.3,E2 -15377.3} C_VEL
LIN {X 0,Y 319.807,Z 247.146,A -85,B 0,C 180,E1 -15381.376,E2 -15381.376} C_VEL
LIN {X 0,Y 319.878,Z 247.136,A -85,B 0,C 180,E1 -15383.695,E2 -15383.695} C_VEL
LIN {X 0,Y 319.948,Z 247.129,A -85,B 0,C 180,E1 -15387.484,E2 -15387.484} C_VEL
LIN {X 0,Y 320.082,Z 247.11,A -85,B 0,C 180,E1 -15390.002,E2 -15390.002} C_VEL
LIN {X 0,Y 319.949,Z 247.128,A -85,B 0,C 180,E1 -15392.52,E2 -15392.52} C_VEL
LIN {X 0,Y 319.88,Z 247.136,A -85,B 0,C 180,E1 -15396.309,E2 -15396.309} C_VEL
LIN {X 0,Y 319.774,Z 247.151,A -85,B 0,C 180,E1 -15398.852,E2 -15398.852} C_VEL
LIN {X 0,Y 319.618,Z 247.168,A -85,B 0,C 180,E1 -15402.704,E2 -15402.704} C_VEL
LIN {X 0,Y 319.619,Z 247.172,A -85,B 0,C 180,E1 -15405.301,E2 -15405.301} C_VEL
LIN {X 0,Y 319.591,Z 247.171,A -85,B 0,C 180,E1 -15409.262,E2 -15409.262} C_VEL
LIN {X 0,Y 319.504,Z 247.184,A -85,B 0,C 180,E1 -15413.326,E2 -15413.326} C_VEL
LIN {X 0,Y 319.579,Z 247.175,A -85,B 0,C 180,E1 -15416.095,E2 -15416.095} C_VEL
LIN {X 0,Y 319.536,Z 247.173,A -85,B 0,C 180,E1 -15418.941,E2 -15418.941} C_VEL
LIN {X 0,Y 319.487,Z 247.187,A -85,B 0,C 180,E1 -15421.869,E2 -15421.869} C_VEL
LIN {X 0,Y 319.531,Z 247.18,A -85,B 0,C 180,E1 -15425.551,E2 -15425.551} C_VEL
LIN {X 0,Y 319.522,Z 247.178,A -85,B 0,C 180,E1 -15429.376,E2 -15429.376} C_VEL
LIN {X 0,Y 318.904,Z 247.263,A -85,B 0,C 180,E1 -15430.428,E2 -15430.428} C_VEL
LIN {X 0,Y 316.075,Z 247.614,A -85,B 0,C 180,E1 -15432.139,E2 -15432.139} C_VEL
LIN {X 0,Y 313.649,Z 247.913,A -85,B 0,C 180,E1 -15433.527,E2 -15433.527} C_VEL
LIN {X 0,Y 312.608,Z 248.046,A -85,B 0,C 180,E1 -15434.601,E2 -15434.601} C_VEL
LIN {X 0,Y 312.525,Z 248.049,A -85,B 0,C 180,E1 -15434.965,E2 -15434.965} C_VEL
LIN {X 0,Y 312.521,Z 248.051,A -85,B 0,C 180,E1 -15437.913,E2 -15437.913} C_VEL
LIN {X 0,Y 312.528,Z 248.051,A -85,B 0,C 180,E1 -15441.914,E2 -15441.914} C_VEL
LIN {X 0,Y 312.48,Z 248.055,A -85,B 0,C 180,E1 -15445.8,E2 -15445.8} C_VEL
LIN {X 0,Y 312.497,Z 248.06,A -85,B 0,C 180,E1 -15448.863,E2 -15448.863} C_VEL
LIN {X 0,Y 312.548,Z 248.049,A -85,B 0,C 180,E1 -15451.834,E2 -15451.834} C_VEL
LIN {X 0,Y 312.567,Z 248.046,A -85,B 0,C 180,E1 -15454.721,E2 -15454.721} C_VEL
LIN {X 0,Y 312.55,Z 248.052,A -85,B 0,C 180,E1 -15457.537,E2 -15457.537} C_VEL
LIN {X 0,Y 312.557,Z 248.05,A -85,B 0,C 180,E1 -15461.662,E2 -15461.662} C_VEL
LIN {X 0,Y 312.68,Z 248.037,A -85,B 0,C 180,E1 -15465.695,E2 -15465.695} C_VEL
LIN {X 0,Y 312.696,Z 248.036,A -85,B 0,C 180,E1 -15469.651,E2 -15469.651} C_VEL
LIN {X 0,Y 312.797,Z 248.017,A -85,B 0,C 180,E1 -15472.261,E2 -15472.261} C_VEL
LIN {X 0,Y 312.698,Z 248.03,A -85,B 0,C 180,E1 -15474.851,E2 -15474.851} C_VEL
LIN {X 0,Y 312.973,Z 247.996,A -85,B 0,C 180,E1 -15478.722,E2 -15478.722} C_VEL
LIN {X 0,Y 312.986,Z 247.993,A -85,B 0,C 180,E1 -15481.295,E2 -15481.295} C_VEL
LIN {X 0,Y 312.852,Z 248.011,A -85,B 0,C 180,E1 -15486.457,E2 -15486.457} C_VEL
LIN {X 0,Y 312.764,Z 248.021,A -85,B 0,C 180,E1 -15489.058,E2 -15489.058} C_VEL
LIN {X 0,Y 312.65,Z 248.038,A -85,B 0,C 180,E1 -15492.998,E2 -15492.998} C_VEL
LIN {X 0,Y 312.639,Z 248.036,A -85,B 0,C 180,E1 -15495.657,E2 -15495.657} C_VEL
LIN {X 0,Y 312.556,Z 248.044,A -85,B 0,C 180,E1 -15499.719,E2 -15499.719} C_VEL
LIN {X 0,Y 312.543,Z 248.054,A -85,B 0,C 180,E1 -15502.784,E2 -15502.784} C_VEL
LIN {X 0,Y 312.55,Z 248.048,A -85,B 0,C 180,E1 -15505.912,E2 -15505.912} C_VEL
LIN {X 0,Y 312.495,Z 248.055,A -85,B 0,C 180,E1 -15509.663,E2 -15509.663} C_VEL
LIN {X 0,Y 312.545,Z 248.051,A -85,B 0,C 180,E1 -15513.693,E2 -15513.693} C_VEL
LIN {X 0,Y 312.535,Z 248.055,A -85,B 0,C 180,E1 -15517.391,E2 -15517.391} C_VEL
LIN {X 0,Y 312.46,Z 248.061,A -85,B 0,C 180,E1 -15520.722,E2 -15520.722} C_VEL
LIN {X 0,Y 312.463,Z 248.061,A -85,B 0,C 180,E1 -15524.216,E2 -15524.216} C_VEL
LIN {X 0,Y 312.452,Z 248.065,A -85,B 0,C 180,E1 -15527.933,E2 -15527.933} C_VEL
LIN {X 0,Y 312.502,Z 248.06,A -85,B 0,C 180,E1 -15531.927,E2 -15531.927} C_VEL
LIN {X 0,Y 312.555,Z 248.052,A -85,B 0,C 180,E1 -15534.221,E2 -15534.221} C_VEL
LIN {X 0,Y 312.528,Z 248.054,A -85,B 0,C 180,E1 -15537.335,E2 -15537.335} C_VEL
LIN {X 0,Y 312.579,Z 248.151,A -85,B 0,C 180,E1 -15539.234,E2 -15539.234} C_VEL
LIN {X 0,Y 314.766,Z 258.827,A -85,B 0,C 180,E1 -15542.678,E2 -15542.678} C_VEL
LIN {X 0,Y 316.361,Z 267.98,A -85,B 0,C 180,E1 -15545.43,E2 -15545.43} C_VEL
LIN {X 0,Y 316.49,Z 269.264,A -85,B 0,C 180,E1 -15545.579,E2 -15545.579} C_VEL
LIN {X 0,Y 322.076,Z 305.574,A -85,B 0,C 180,E1 -15546.912,E2 -15546.912} C_VEL
LIN {X 0,Y 320.226,Z 375.875,A -85,B 0,C 180,E1 -15548.641,E2 -15548.641} C_VEL
LIN {X 0,Y 319.474,Z 389.562,A -85,B 0,C 180,E1 -15549.221,E2 -15549.221} C_VEL
LIN {X 0,Y 318.544,Z 402.046,A -85,B 0,C 180,E1 -15550.001,E2 -15550.001} C_VEL
LIN {X 0,Y 317.479,Z 413.268,A -85,B 0,C 180,E1 -15550.94,E2 -15550.94} C_VEL
LIN {X 0,Y 316.189,Z 424.941,A -85,B 0,C 180,E1 -15552.202,E2 -15552.202} C_VEL
LIN {X 0,Y 315.079,Z 435.084,A -85,B 0,C 180,E1 -15553.58,E2 -15553.58} C_VEL
LIN {X 0,Y 313.989,Z 444.103,A -85,B 0,C 180,E1 -15555.082,E2 -15555.082} C_VEL
LIN {X 0,Y 313.011,Z 452.033,A -85,B 0,C 180,E1 -15556.693,E2 -15556.693} C_VEL
LIN {X 0,Y 312.055,Z 459.755,A -85,B 0,C 180,E1 -15558.633,E2 -15558.633} C_VEL
LIN {X 0,Y 311.527,Z 465.031,A -85,B 0,C 180,E1 -15560.257,E2 -15560.257} C_VEL
LIN {X 0,Y 311.058,Z 470.12,A -85,B 0,C 180,E1 -15562.207,E2 -15562.207} C_VEL
LIN {X 0,Y 310.799,Z 474.255,A -85,B 0,C 180,E1 -15564.289,E2 -15564.289} C_VEL
LIN {X 0,Y 310.702,Z 476.889,A -85,B 0,C 180,E1 -15566.107,E2 -15566.107} C_VEL
LIN {X 0,Y 310.666,Z 478.226,A -85,B 0,C 180,E1 -15567.405,E2 -15567.405} C_VEL
LIN {X 0,Y 310.621,Z 479.157,A -85,B 0,C 180,E1 -15568.701,E2 -15568.701} C_VEL
LIN {X 0,Y 310.63,Z 479.675,A -85,B 0,C 180,E1 -15569.998,E2 -15569.998} C_VEL
LIN {X 0,Y 310.619,Z 479.747,A -85,B 0,C 180,E1 -15571.294,E2 -15571.294} C_VEL
LIN {X 0,Y 310.665,Z 479.423,A -85,B 0,C 180,E1 -15572.591,E2 -15572.591} C_VEL
LIN {X 0,Y 310.707,Z 478.705,A -85,B 0,C 180,E1 -15573.889,E2 -15573.889} C_VEL
LIN {X 0,Y 310.797,Z 476.979,A -85,B 0,C 180,E1 -15575.707,E2 -15575.707} C_VEL
LIN {X 0,Y 311.142,Z 473.993,A -85,B 0,C 180,E1 -15577.787,E2 -15577.787} C_VEL
LIN {X 0,Y 311.71,Z 470.128,A -85,B 0,C 180,E1 -15579.733,E2 -15579.733} C_VEL
LIN {X 0,Y 312.523,Z 465.135,A -85,B 0,C 180,E1 -15581.674,E2 -15581.674} C_VEL
LIN {X 0,Y 313.597,Z 458.868,A -85,B 0,C 180,E1 -15583.608,E2 -15583.608} C_VEL
LIN {X 0,Y 315.158,Z 451.057,A -85,B 0,C 180,E1 -15585.519,E2 -15585.519} C_VEL
LIN {X 0,Y 316.708,Z 441.52,A -85,B 0,C 180,E1 -15587.392,E2 -15587.392} C_VEL
LIN {X 0,Y 318.397,Z 431.276,A -85,B 0,C 180,E1 -15588.998,E2 -15588.998} C_VEL
LIN {X 0,Y 320.203,Z 419.969,A -85,B 0,C 180,E1 -15590.389,E2 -15590.389} C_VEL
LIN {X 0,Y 321.638,Z 409.008,A -85,B 0,C 180,E1 -15591.466,E2 -15591.466} C_VEL
